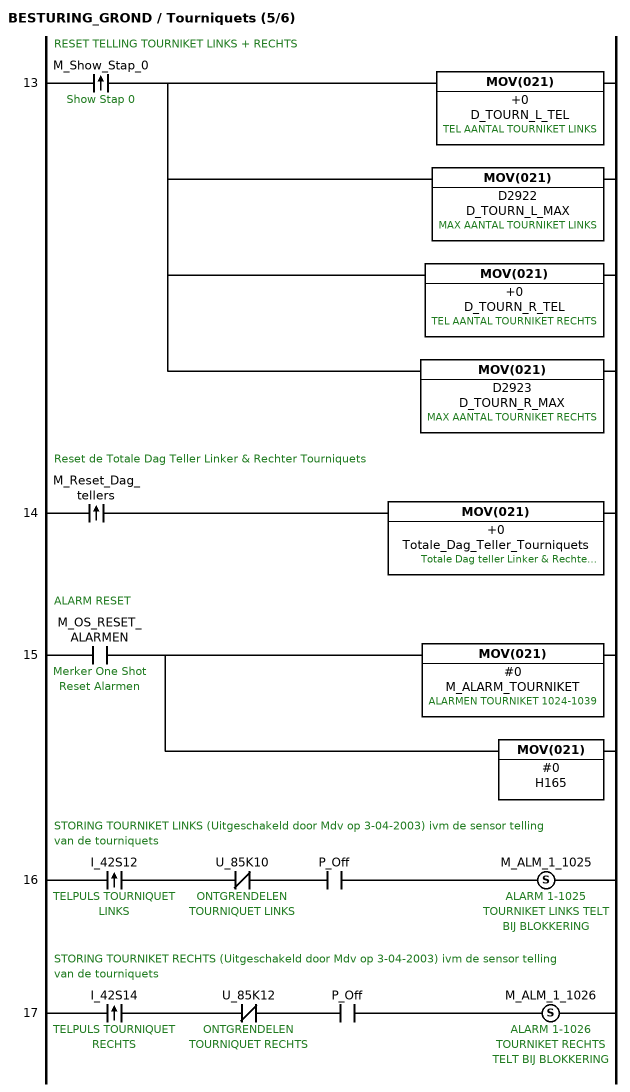
; [picture p144: BESTURING_GROND / Tourniquets, rungs 13-17]
; rung 13: RESET TELLING TOURNIKET LINKS + RECHTS
@LD M_Show_Stap_0  ; Show Stap 0
MOV(021) +0 D_TOURN_L_TEL  ; TEL AANTAL TOURNIKET LINKS
MOV(021) D2922 D_TOURN_L_MAX  ; MAX AANTAL TOURNIKET LINKS
MOV(021) +0 D_TOURN_R_TEL  ; TEL AANTAL TOURNIKET RECHTS
MOV(021) D2923 D_TOURN_R_MAX  ; MAX AANTAL TOURNIKET RECHTS
; rung 14: Reset de Totale Dag Teller Linker & Rechter Tourniquets
@LD M_Reset_Dag_tellers
MOV(021) +0 Totale_Dag_Teller_Tourniquets  ; Totale Dag teller Linker & Rechter Tournoquets
; rung 15: ALARM RESET
LD M_OS_RESET_ALARMEN  ; Merker One Shot Reset Alarmen
MOV(021) #0 M_ALARM_TOURNIKET  ; ALARMEN TOURNIKET 1024-1039
MOV(021) #0 H165
; rung 16: STORING TOURNIKET LINKS (Uitgeschakeld door Mdv op 3-04-2003) ivm de sensor telling van de tourniquets
@LD I_42S12  ; TELPULS TOURNIQUET LINKS
ANDNOT U_85K10  ; ONTGRENDELEN TOURNIQUET LINKS
AND P_Off
SET M_ALM_1_1025  ; ALARM 1-1025 TOURNIKET LINKS TELT BIJ BLOKKERING
; rung 17: STORING TOURNIKET RECHTS (Uitgeschakeld door Mdv op 3-04-2003) ivm de sensor telling van de tourniquets
@LD I_42S14  ; TELPULS TOURNIQUET RECHTS
ANDNOT U_85K12  ; ONTGRENDELEN TOURNIQUET RECHTS
AND P_Off
SET M_ALM_1_1026  ; ALARM 1-1026 TOURNIKET RECHTS TELT BIJ BLOKKERING

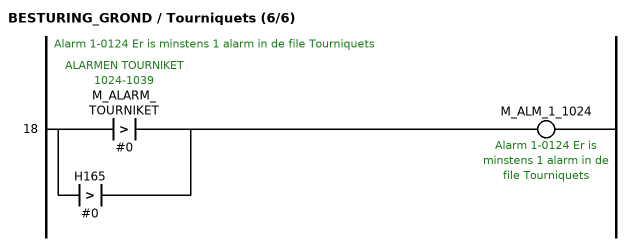
; rung 18: Alarm 1-0124 Er is minstens 1 alarm in de file Tourniquets
LD>(320) M_ALARM_TOURNIKET #0  ; ALARMEN TOURNIKET 1024-1039
OR>(320) H165 #0
OUT M_ALM_1_1024  ; Alarm 1-0124 Er is minstens 1 alarm in de file Tourniquets

### Section Hydaruliek_Arm

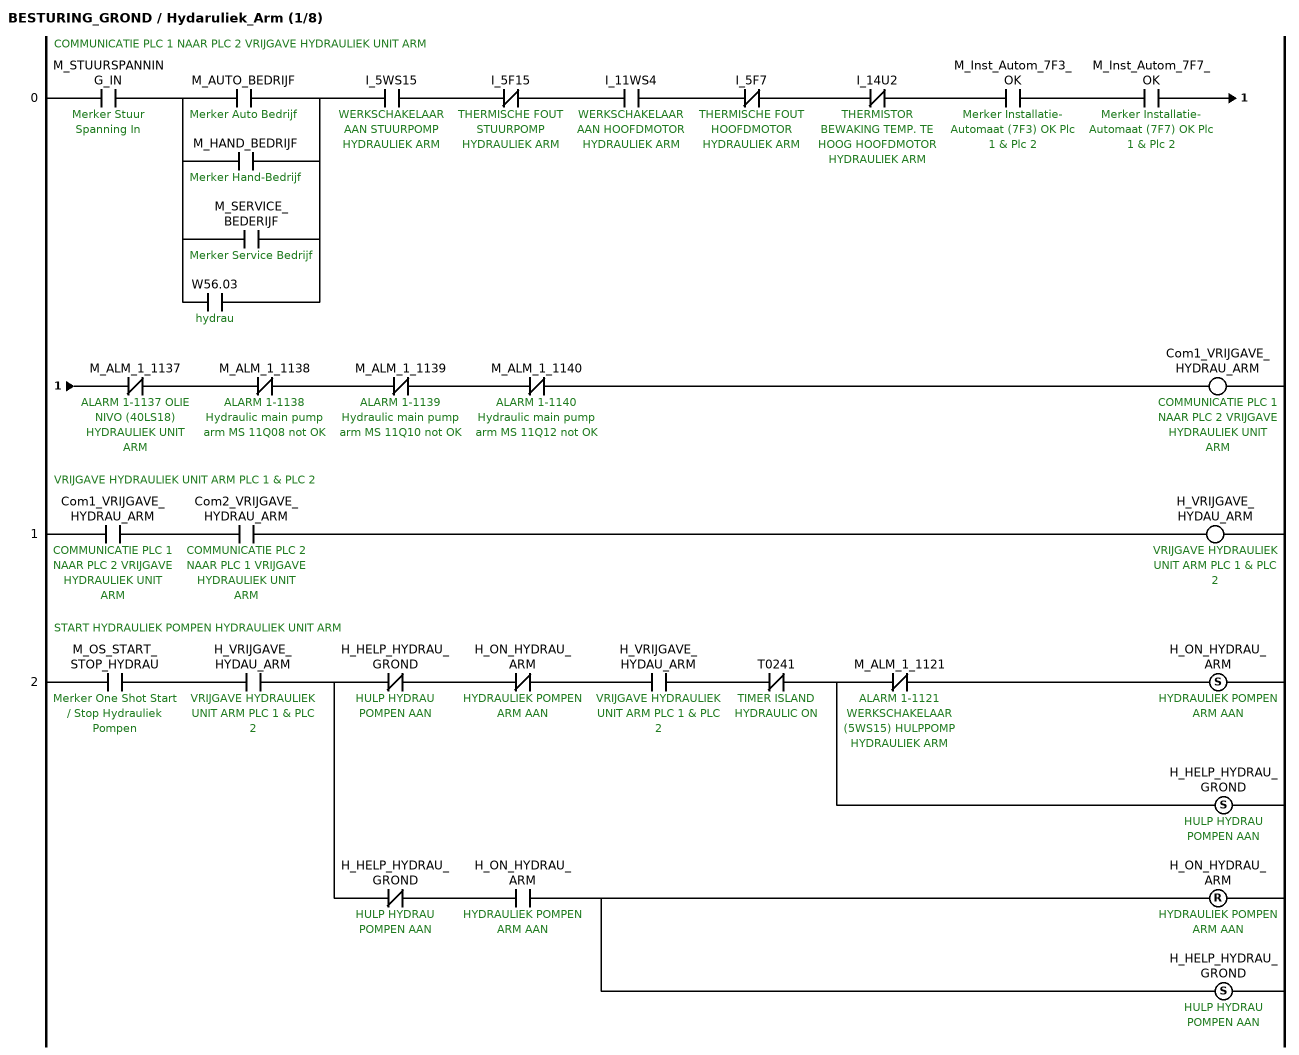
; rung 0: COMMUNICATIE PLC 1 NAAR PLC 2 VRIJGAVE HYDRAULIEK UNIT ARM
LD M_STUURSPANNING_IN  ; Merker Stuur Spanning In
LD M_AUTO_BEDRIJF  ; Merker Auto Bedrijf
OR M_HAND_BEDRIJF  ; Merker Hand-Bedrijf
OR M_SERVICE_BEDERIJF  ; Merker Service Bedrijf
OR W56.03  ; hydrau
ANDLD
AND I_5WS15  ; WERKSCHAKELAAR AAN STUURPOMP HYDRAULIEK ARM
ANDNOT I_5F15  ; THERMISCHE FOUT STUURPOMP HYDRAULIEK ARM
AND I_11WS4  ; WERKSCHAKELAAR AAN HOOFDMOTOR HYDRAULIEK ARM
ANDNOT I_5F7  ; THERMISCHE FOUT HOOFDMOTOR HYDRAULIEK ARM
ANDNOT I_14U2  ; THERMISTOR BEWAKING TEMP. TE HOOG HOOFDMOTOR HYDRAULIEK ARM
AND M_Inst_Autom_7F3_OK  ; Merker Installatie-Automaat (7F3) OK Plc 1 & Plc 2
AND M_Inst_Autom_7F7_OK  ; Merker Installatie-Automaat (7F7) OK Plc 1 & Plc 2
ANDNOT M_ALM_1_1137  ; ALARM 1-1137 OLIE NIVO (40LS18) HYDRAULIEK UNIT ARM
ANDNOT M_ALM_1_1138  ; ALARM 1-1138 Hydraulic main pump arm MS 11Q08 not OK
ANDNOT M_ALM_1_1139  ; ALARM 1-1139 Hydraulic main pump arm MS 11Q10 not OK
ANDNOT M_ALM_1_1140  ; ALARM 1-1140 Hydraulic main pump arm MS 11Q12 not OK
OUT Com1_VRIJGAVE_HYDRAU_ARM  ; COMMUNICATIE PLC 1 NAAR PLC 2 VRIJGAVE HYDRAULIEK UNIT ARM
; rung 1: VRIJGAVE HYDRAULIEK UNIT ARM PLC 1 & PLC 2
LD Com1_VRIJGAVE_HYDRAU_ARM  ; COMMUNICATIE PLC 1 NAAR PLC 2 VRIJGAVE HYDRAULIEK UNIT ARM
AND Com2_VRIJGAVE_HYDRAU_ARM  ; COMMUNICATIE PLC 2 NAAR PLC 1 VRIJGAVE HYDRAULIEK UNIT ARM
OUT H_VRIJGAVE_HYDAU_ARM  ; VRIJGAVE HYDRAULIEK UNIT ARM PLC 1 & PLC 2
; rung 2: START HYDRAULIEK POMPEN HYDRAULIEK UNIT ARM
LD M_OS_START_STOP_HYDRAU  ; Merker One Shot Start / Stop Hydrauliek Pompen
AND H_VRIJGAVE_HYDAU_ARM  ; VRIJGAVE HYDRAULIEK UNIT ARM PLC 1 & PLC 2
OUT TR0
ANDNOT H_HELP_HYDRAU_GROND  ; HULP HYDRAU POMPEN AAN
ANDNOT H_ON_HYDRAU_ARM  ; HYDRAULIEK POMPEN ARM AAN
AND H_VRIJGAVE_HYDAU_ARM  ; VRIJGAVE HYDRAULIEK UNIT ARM PLC 1 & PLC 2
ANDNOT T0241  ; TIMER ISLAND HYDRAULIC ON
OUT TR1
ANDNOT M_ALM_1_1121  ; ALARM 1-1121 WERKSCHAKELAAR (5WS15) HULPPOMP HYDRAULIEK ARM
SET H_ON_HYDRAU_ARM  ; HYDRAULIEK POMPEN ARM AAN
LD TR1
SET H_HELP_HYDRAU_GROND  ; HULP HYDRAU POMPEN AAN
LD TR0
ANDNOT H_HELP_HYDRAU_GROND  ; HULP HYDRAU POMPEN AAN
AND H_ON_HYDRAU_ARM  ; HYDRAULIEK POMPEN ARM AAN
RSET H_ON_HYDRAU_ARM  ; HYDRAULIEK POMPEN ARM AAN
SET H_HELP_HYDRAU_GROND  ; HULP HYDRAU POMPEN AAN

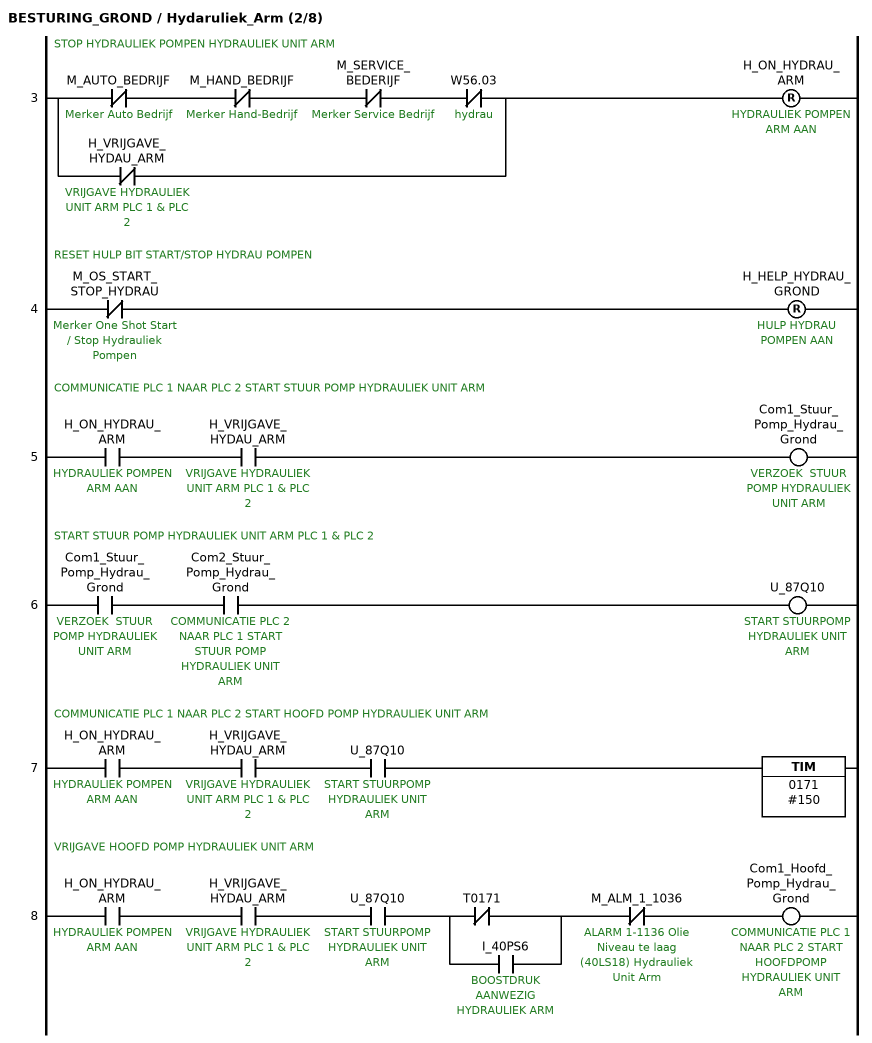
; rung 3: STOP HYDRAULIEK POMPEN HYDRAULIEK UNIT ARM
LDNOT M_AUTO_BEDRIJF  ; Merker Auto Bedrijf
ANDNOT M_HAND_BEDRIJF  ; Merker Hand-Bedrijf
ANDNOT M_SERVICE_BEDERIJF  ; Merker Service Bedrijf
ANDNOT W56.03  ; hydrau
ORNOT H_VRIJGAVE_HYDAU_ARM  ; VRIJGAVE HYDRAULIEK UNIT ARM PLC 1 & PLC 2
RSET H_ON_HYDRAU_ARM  ; HYDRAULIEK POMPEN ARM AAN
; rung 4: RESET HULP BIT START/STOP HYDRAU POMPEN
LDNOT M_OS_START_STOP_HYDRAU  ; Merker One Shot Start / Stop Hydrauliek Pompen
RSET H_HELP_HYDRAU_GROND  ; HULP HYDRAU POMPEN AAN
; rung 5: COMMUNICATIE PLC 1 NAAR PLC 2 START STUUR POMP HYDRAULIEK UNIT ARM
LD H_ON_HYDRAU_ARM  ; HYDRAULIEK POMPEN ARM AAN
AND H_VRIJGAVE_HYDAU_ARM  ; VRIJGAVE HYDRAULIEK UNIT ARM PLC 1 & PLC 2
OUT Com1_Stuur_Pomp_Hydrau_Grond  ; VERZOEK  STUUR POMP HYDRAULIEK UNIT ARM
; rung 6: START STUUR POMP HYDRAULIEK UNIT ARM PLC 1 & PLC 2
LD Com1_Stuur_Pomp_Hydrau_Grond  ; VERZOEK  STUUR POMP HYDRAULIEK UNIT ARM
AND Com2_Stuur_Pomp_Hydrau_Grond  ; COMMUNICATIE PLC 2 NAAR PLC 1 START STUUR POMP HYDRAULIEK UNIT ARM
OUT U_87Q10  ; START STUURPOMP HYDRAULIEK UNIT ARM
; rung 7: COMMUNICATIE PLC 1 NAAR PLC 2 START HOOFD POMP HYDRAULIEK UNIT ARM
LD H_ON_HYDRAU_ARM  ; HYDRAULIEK POMPEN ARM AAN
AND H_VRIJGAVE_HYDAU_ARM  ; VRIJGAVE HYDRAULIEK UNIT ARM PLC 1 & PLC 2
AND U_87Q10  ; START STUURPOMP HYDRAULIEK UNIT ARM
TIM 0171 #150
; rung 8: VRIJGAVE HOOFD POMP HYDRAULIEK UNIT ARM
LD H_ON_HYDRAU_ARM  ; HYDRAULIEK POMPEN ARM AAN
AND H_VRIJGAVE_HYDAU_ARM  ; VRIJGAVE HYDRAULIEK UNIT ARM PLC 1 & PLC 2
AND U_87Q10  ; START STUURPOMP HYDRAULIEK UNIT ARM
LDNOT T0171
OR I_40PS6  ; BOOSTDRUK AANWEZIG HYDRAULIEK ARM
ANDLD
ANDNOT M_ALM_1_1036  ; ALARM 1-1136 Olie Niveau te laag (40LS18) Hydrauliek Unit Arm
OUT Com1_Hoofd_Pomp_Hydrau_Grond  ; COMMUNICATIE PLC 1 NAAR PLC 2 START HOOFDPOMP HYDRAULIEK UNIT ARM

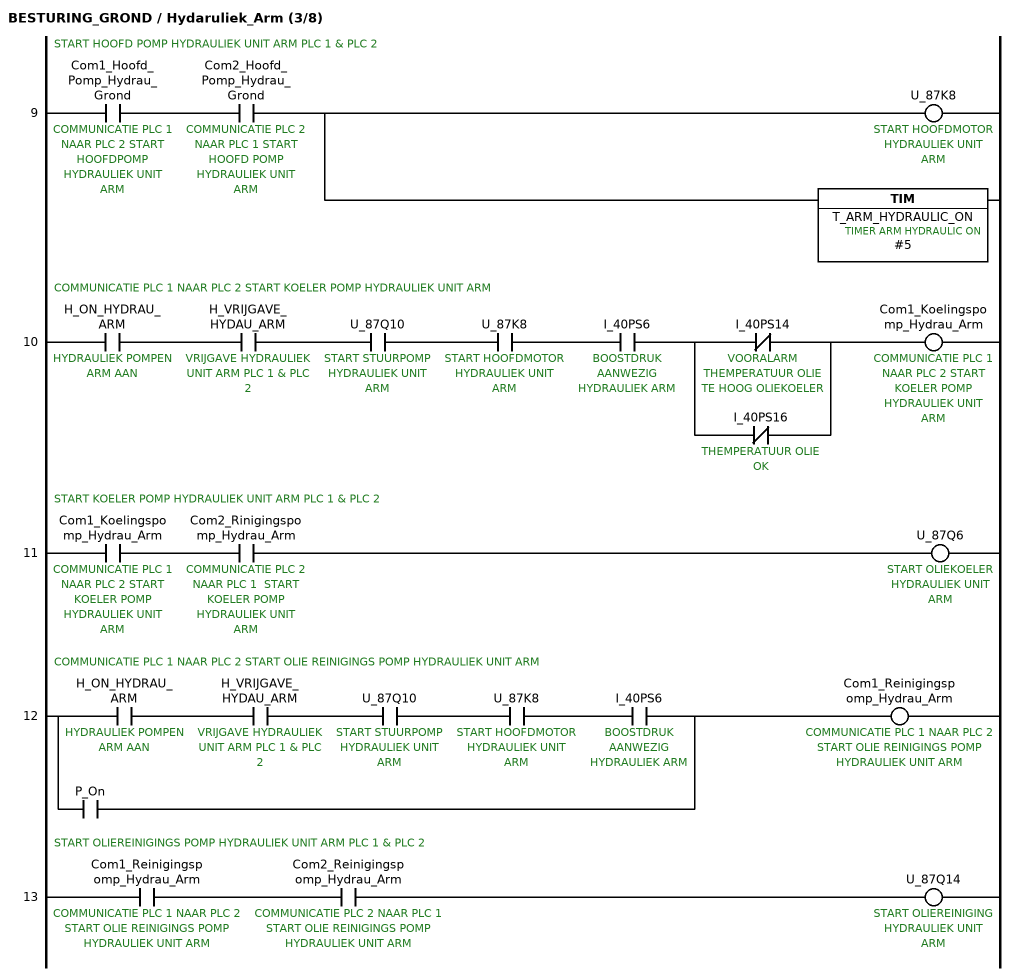
; rung 9: START HOOFD POMP HYDRAULIEK UNIT ARM PLC 1 & PLC 2
LD Com1_Hoofd_Pomp_Hydrau_Grond  ; COMMUNICATIE PLC 1 NAAR PLC 2 START HOOFDPOMP HYDRAULIEK UNIT ARM
AND Com2_Hoofd_Pomp_Hydrau_Grond  ; COMMUNICATIE PLC 2 NAAR PLC 1 START HOOFD POMP HYDRAULIEK UNIT ARM
OUT U_87K8  ; START HOOFDMOTOR HYDRAULIEK UNIT ARM
TIM T_ARM_HYDRAULIC_ON #5  ; TIMER ARM HYDRAULIC ON
; rung 10: COMMUNICATIE PLC 1 NAAR PLC 2 START KOELER POMP HYDRAULIEK UNIT ARM
LD H_ON_HYDRAU_ARM  ; HYDRAULIEK POMPEN ARM AAN
AND H_VRIJGAVE_HYDAU_ARM  ; VRIJGAVE HYDRAULIEK UNIT ARM PLC 1 & PLC 2
AND U_87Q10  ; START STUURPOMP HYDRAULIEK UNIT ARM
AND U_87K8  ; START HOOFDMOTOR HYDRAULIEK UNIT ARM
AND I_40PS6  ; BOOSTDRUK AANWEZIG HYDRAULIEK ARM
LDNOT I_40PS14  ; VOORALARM THEMPERATUUR OLIE TE HOOG OLIEKOELER
ORNOT I_40PS16  ; THEMPERATUUR OLIE OK
ANDLD
OUT Com1_Koelingspomp_Hydrau_Arm  ; COMMUNICATIE PLC 1 NAAR PLC 2 START KOELER POMP HYDRAULIEK UNIT ARM
; rung 11: START KOELER POMP HYDRAULIEK UNIT ARM PLC 1 & PLC 2
LD Com1_Koelingspomp_Hydrau_Arm  ; COMMUNICATIE PLC 1 NAAR PLC 2 START KOELER POMP HYDRAULIEK UNIT ARM
AND Com2_Rinigingspomp_Hydrau_Arm  ; COMMUNICATIE PLC 2 NAAR PLC 1  START KOELER POMP HYDRAULIEK UNIT ARM
OUT U_87Q6  ; START OLIEKOELER HYDRAULIEK UNIT ARM
; rung 12: COMMUNICATIE PLC 1 NAAR PLC 2 START OLIE REINIGINGS POMP HYDRAULIEK UNIT ARM
LD H_ON_HYDRAU_ARM  ; HYDRAULIEK POMPEN ARM AAN
AND H_VRIJGAVE_HYDAU_ARM  ; VRIJGAVE HYDRAULIEK UNIT ARM PLC 1 & PLC 2
AND U_87Q10  ; START STUURPOMP HYDRAULIEK UNIT ARM
AND U_87K8  ; START HOOFDMOTOR HYDRAULIEK UNIT ARM
AND I_40PS6  ; BOOSTDRUK AANWEZIG HYDRAULIEK ARM
OR P_On
OUT Com1_Reinigingspomp_Hydrau_Arm  ; COMMUNICATIE PLC 1 NAAR PLC 2 START OLIE REINIGINGS POMP HYDRAULIEK UNIT ARM
; rung 13: START OLIEREINIGINGS POMP HYDRAULIEK UNIT ARM PLC 1 & PLC 2
LD Com1_Reinigingspomp_Hydrau_Arm  ; COMMUNICATIE PLC 1 NAAR PLC 2 START OLIE REINIGINGS POMP HYDRAULIEK UNIT ARM
AND Com2_Reinigingspomp_Hydrau_Arm  ; COMMUNICATIE PLC 2 NAAR PLC 1 START OLIE REINIGINGS POMP HYDRAULIEK UNIT ARM
OUT U_87Q14  ; START OLIEREINIGING HYDRAULIEK UNIT ARM

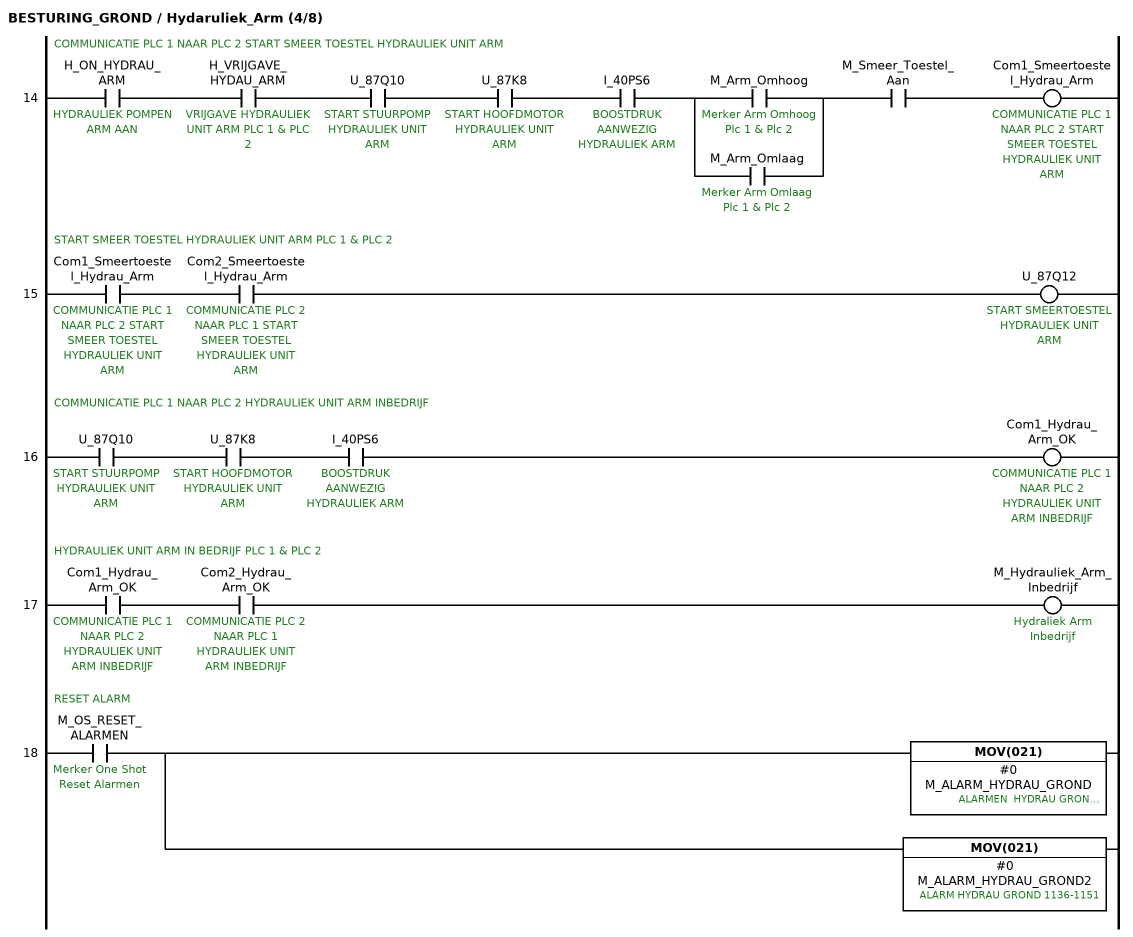
; rung 14: COMMUNICATIE PLC 1 NAAR PLC 2 START SMEER TOESTEL HYDRAULIEK UNIT ARM
LD H_ON_HYDRAU_ARM  ; HYDRAULIEK POMPEN ARM AAN
AND H_VRIJGAVE_HYDAU_ARM  ; VRIJGAVE HYDRAULIEK UNIT ARM PLC 1 & PLC 2
AND U_87Q10  ; START STUURPOMP HYDRAULIEK UNIT ARM
AND U_87K8  ; START HOOFDMOTOR HYDRAULIEK UNIT ARM
AND I_40PS6  ; BOOSTDRUK AANWEZIG HYDRAULIEK ARM
LD M_Arm_Omhoog  ; Merker Arm Omhoog Plc 1 & Plc 2
OR M_Arm_Omlaag  ; Merker Arm Omlaag Plc 1 & Plc 2
ANDLD
AND M_Smeer_Toestel_Aan
OUT Com1_Smeertoestel_Hydrau_Arm  ; COMMUNICATIE PLC 1 NAAR PLC 2 START SMEER TOESTEL HYDRAULIEK UNIT ARM
; rung 15: START SMEER TOESTEL HYDRAULIEK UNIT ARM PLC 1 & PLC 2
LD Com1_Smeertoestel_Hydrau_Arm  ; COMMUNICATIE PLC 1 NAAR PLC 2 START SMEER TOESTEL HYDRAULIEK UNIT ARM
AND Com2_Smeertoestel_Hydrau_Arm  ; COMMUNICATIE PLC 2 NAAR PLC 1 START SMEER TOESTEL HYDRAULIEK UNIT ARM
OUT U_87Q12  ; START SMEERTOESTEL HYDRAULIEK UNIT ARM
; rung 16: COMMUNICATIE PLC 1 NAAR PLC 2 HYDRAULIEK UNIT ARM INBEDRIJF
LD U_87Q10  ; START STUURPOMP HYDRAULIEK UNIT ARM
AND U_87K8  ; START HOOFDMOTOR HYDRAULIEK UNIT ARM
AND I_40PS6  ; BOOSTDRUK AANWEZIG HYDRAULIEK ARM
OUT Com1_Hydrau_Arm_OK  ; COMMUNICATIE PLC 1 NAAR PLC 2 HYDRAULIEK UNIT ARM INBEDRIJF
; rung 17: HYDRAULIEK UNIT ARM IN BEDRIJF PLC 1 & PLC 2
LD Com1_Hydrau_Arm_OK  ; COMMUNICATIE PLC 1 NAAR PLC 2 HYDRAULIEK UNIT ARM INBEDRIJF
AND Com2_Hydrau_Arm_OK  ; COMMUNICATIE PLC 2 NAAR PLC 1 HYDRAULIEK UNIT ARM INBEDRIJF
OUT M_Hydrauliek_Arm_Inbedrijf  ; Hydraliek Arm Inbedrijf
; rung 18: RESET ALARM
LD M_OS_RESET_ALARMEN  ; Merker One Shot Reset Alarmen
MOV(021) #0 M_ALARM_HYDRAU_GROND  ; ALARMEN  HYDRAU GROND 1120-1135
MOV(021) #0 M_ALARM_HYDRAU_GROND2  ; ALARM HYDRAU GROND 1136-1151

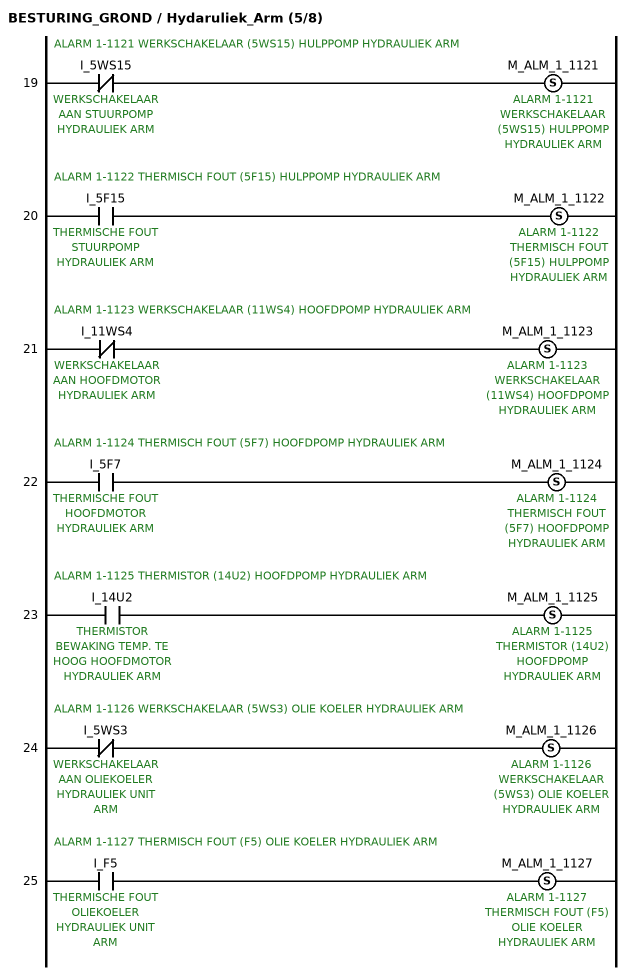
; rung 19: ALARM 1-1121 WERKSCHAKELAAR (5WS15) HULPPOMP HYDRAULIEK ARM
LDNOT I_5WS15  ; WERKSCHAKELAAR AAN STUURPOMP HYDRAULIEK ARM
SET M_ALM_1_1121  ; ALARM 1-1121 WERKSCHAKELAAR (5WS15) HULPPOMP HYDRAULIEK ARM
; rung 20: ALARM 1-1122 THERMISCH FOUT (5F15) HULPPOMP HYDRAULIEK ARM
LD I_5F15  ; THERMISCHE FOUT STUURPOMP HYDRAULIEK ARM
SET M_ALM_1_1122  ; ALARM 1-1122 THERMISCH FOUT (5F15) HULPPOMP HYDRAULIEK ARM
; rung 21: ALARM 1-1123 WERKSCHAKELAAR (11WS4) HOOFDPOMP HYDRAULIEK ARM
LDNOT I_11WS4  ; WERKSCHAKELAAR AAN HOOFDMOTOR HYDRAULIEK ARM
SET M_ALM_1_1123  ; ALARM 1-1123 WERKSCHAKELAAR (11WS4) HOOFDPOMP HYDRAULIEK ARM
; rung 22: ALARM 1-1124 THERMISCH FOUT (5F7) HOOFDPOMP HYDRAULIEK ARM
LD I_5F7  ; THERMISCHE FOUT HOOFDMOTOR HYDRAULIEK ARM
SET M_ALM_1_1124  ; ALARM 1-1124 THERMISCH FOUT (5F7) HOOFDPOMP HYDRAULIEK ARM
; rung 23: ALARM 1-1125 THERMISTOR (14U2) HOOFDPOMP HYDRAULIEK ARM
LD I_14U2  ; THERMISTOR BEWAKING TEMP. TE HOOG HOOFDMOTOR HYDRAULIEK ARM
SET M_ALM_1_1125  ; ALARM 1-1125 THERMISTOR (14U2) HOOFDPOMP HYDRAULIEK ARM
; rung 24: ALARM 1-1126 WERKSCHAKELAAR (5WS3) OLIE KOELER HYDRAULIEK ARM
LDNOT I_5WS3  ; WERKSCHAKELAAR AAN OLIEKOELER HYDRAULIEK UNIT ARM
SET M_ALM_1_1126  ; ALARM 1-1126 WERKSCHAKELAAR (5WS3) OLIE KOELER HYDRAULIEK ARM
; rung 25: ALARM 1-1127 THERMISCH FOUT (F5) OLIE KOELER HYDRAULIEK ARM
LD I_F5  ; THERMISCHE FOUT OLIEKOELER HYDRAULIEK UNIT ARM
SET M_ALM_1_1127  ; ALARM 1-1127 THERMISCH FOUT (F5) OLIE KOELER HYDRAULIEK ARM

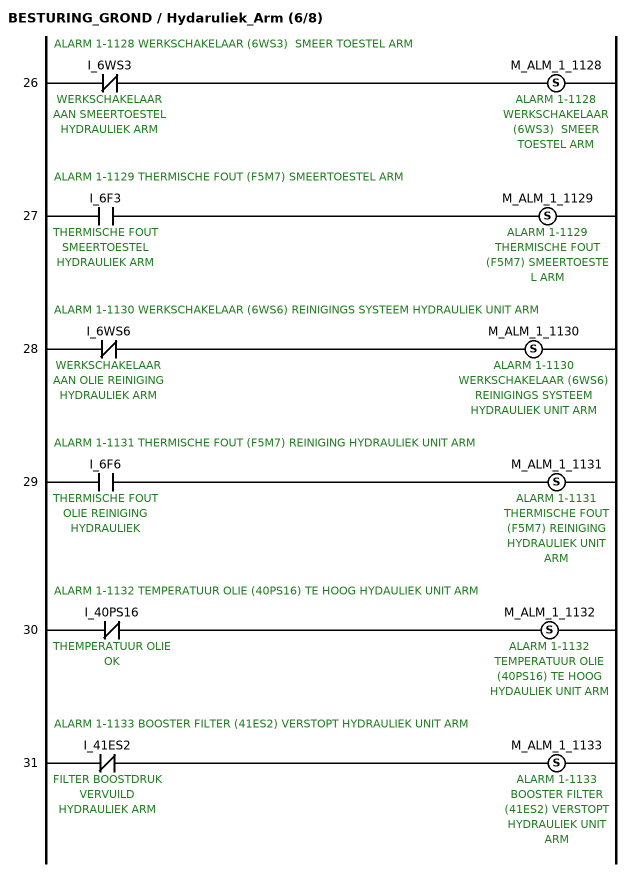
; rung 26: ALARM 1-1128 WERKSCHAKELAAR (6WS3)  SMEER TOESTEL ARM
LDNOT I_6WS3  ; WERKSCHAKELAAR AAN SMEERTOESTEL HYDRAULIEK ARM
SET M_ALM_1_1128  ; ALARM 1-1128 WERKSCHAKELAAR (6WS3)  SMEER TOESTEL ARM
; rung 27: ALARM 1-1129 THERMISCHE FOUT (F5M7) SMEERTOESTEL ARM
LD I_6F3  ; THERMISCHE FOUT SMEERTOESTEL HYDRAULIEK ARM
SET M_ALM_1_1129  ; ALARM 1-1129 THERMISCHE FOUT (F5M7) SMEERTOESTEL ARM
; rung 28: ALARM 1-1130 WERKSCHAKELAAR (6WS6) REINIGINGS SYSTEEM HYDRAULIEK UNIT ARM
LDNOT I_6WS6  ; WERKSCHAKELAAR AAN OLIE REINIGING HYDRAULIEK ARM
SET M_ALM_1_1130  ; ALARM 1-1130 WERKSCHAKELAAR (6WS6) REINIGINGS SYSTEEM HYDRAULIEK UNIT ARM
; rung 29: ALARM 1-1131 THERMISCHE FOUT (F5M7) REINIGING HYDRAULIEK UNIT ARM
LD I_6F6  ; THERMISCHE FOUT OLIE REINIGING HYDRAULIEK
SET M_ALM_1_1131  ; ALARM 1-1131 THERMISCHE FOUT (F5M7) REINIGING HYDRAULIEK UNIT ARM
; rung 30: ALARM 1-1132 TEMPERATUUR OLIE (40PS16) TE HOOG HYDAULIEK UNIT ARM
LDNOT I_40PS16  ; THEMPERATUUR OLIE OK
SET M_ALM_1_1132  ; ALARM 1-1132 TEMPERATUUR OLIE (40PS16) TE HOOG HYDAULIEK UNIT ARM
; rung 31: ALARM 1-1133 BOOSTER FILTER (41ES2) VERSTOPT HYDRAULIEK UNIT ARM
LDNOT I_41ES2  ; FILTER BOOSTDRUK VERVUILD HYDRAULIEK ARM
SET M_ALM_1_1133  ; ALARM 1-1133 BOOSTER FILTER (41ES2) VERSTOPT HYDRAULIEK UNIT ARM

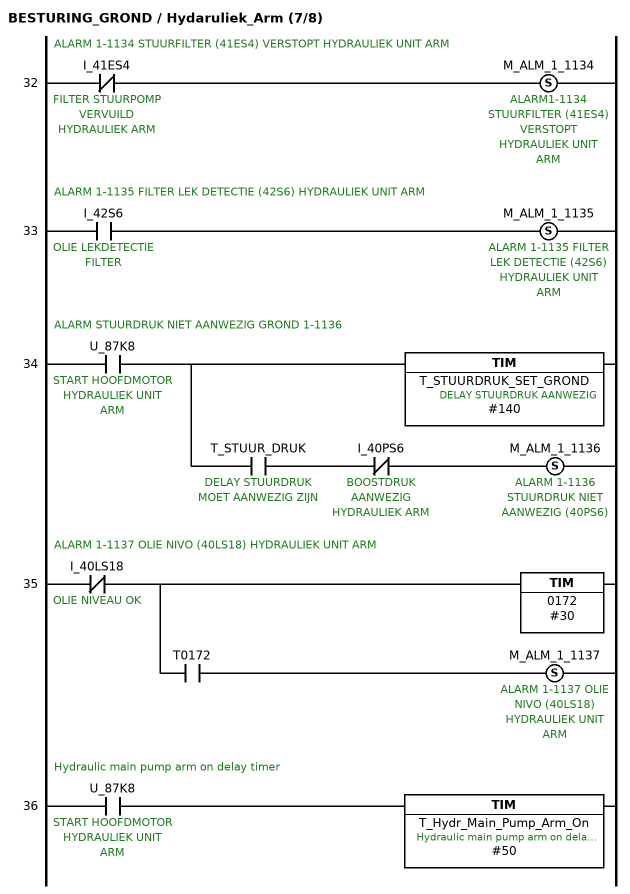
; rung 32: ALARM 1-1134 STUURFILTER (41ES4) VERSTOPT HYDRAULIEK UNIT ARM
LDNOT I_41ES4  ; FILTER STUURPOMP VERVUILD HYDRAULIEK ARM
SET M_ALM_1_1134  ; ALARM1-1134 STUURFILTER (41ES4) VERSTOPT HYDRAULIEK UNIT ARM
; rung 33: ALARM 1-1135 FILTER LEK DETECTIE (42S6) HYDRAULIEK UNIT ARM
LD I_42S6  ; OLIE LEKDETECTIE FILTER
SET M_ALM_1_1135  ; ALARM 1-1135 FILTER LEK DETECTIE (42S6) HYDRAULIEK UNIT ARM
; rung 34: ALARM STUURDRUK NIET AANWEZIG GROND 1-1136
LD U_87K8  ; START HOOFDMOTOR HYDRAULIEK UNIT ARM
TIM T_STUURDRUK_SET_GROND #140  ; DELAY STUURDRUK AANWEZIG
AND T_STUUR_DRUK  ; DELAY STUURDRUK MOET AANWEZIG ZIJN
ANDNOT I_40PS6  ; BOOSTDRUK AANWEZIG HYDRAULIEK ARM
SET M_ALM_1_1136  ; ALARM 1-1136 STUURDRUK NIET AANWEZIG (40PS6)
; rung 35: ALARM 1-1137 OLIE NIVO (40LS18) HYDRAULIEK UNIT ARM
LDNOT I_40LS18  ; OLIE NIVEAU OK
TIM 0172 #30
AND T0172
SET M_ALM_1_1137  ; ALARM 1-1137 OLIE NIVO (40LS18) HYDRAULIEK UNIT ARM
; rung 36: Hydraulic main pump arm on delay timer
LD U_87K8  ; START HOOFDMOTOR HYDRAULIEK UNIT ARM
TIM T_Hydr_Main_Pump_Arm_On #50  ; Hydraulic main pump arm on delay timer

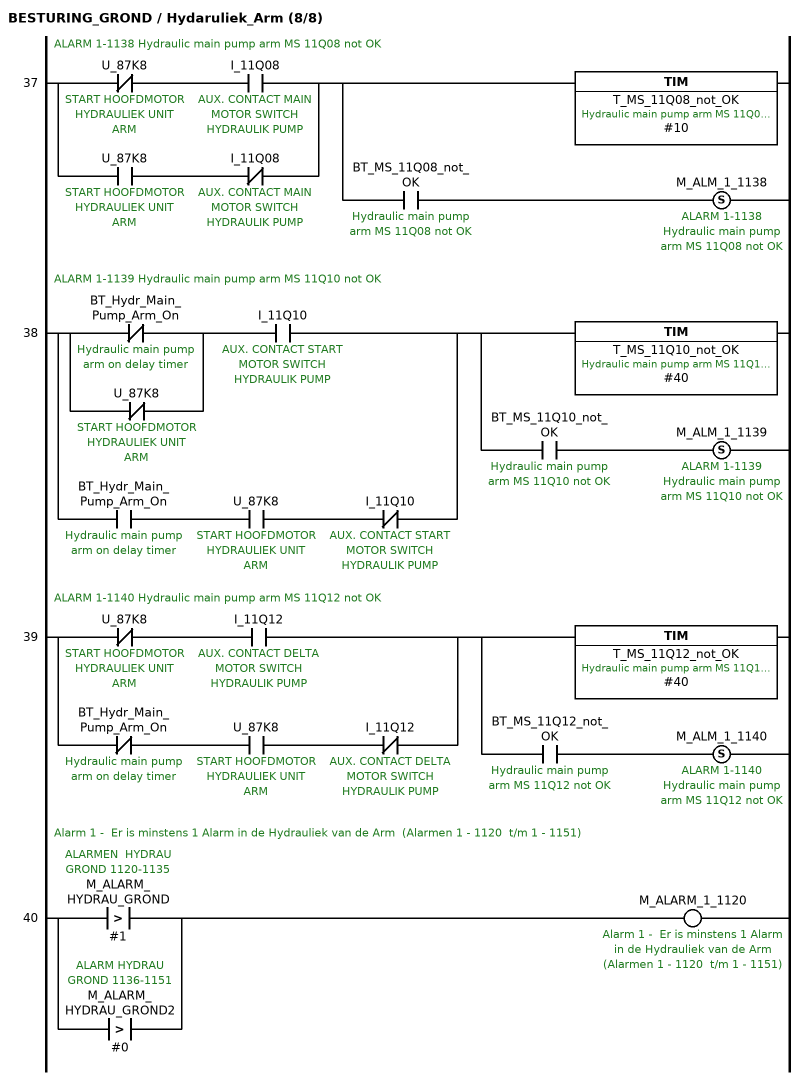
; rung 37: ALARM 1-1138 Hydraulic main pump arm MS 11Q08 not OK
LDNOT U_87K8  ; START HOOFDMOTOR HYDRAULIEK UNIT ARM
AND I_11Q08  ; AUX. CONTACT MAIN MOTOR SWITCH HYDRAULIK PUMP
LD U_87K8  ; START HOOFDMOTOR HYDRAULIEK UNIT ARM
ANDNOT I_11Q08  ; AUX. CONTACT MAIN MOTOR SWITCH HYDRAULIK PUMP
ORLD
TIM T_MS_11Q08_not_OK #10  ; Hydraulic main pump arm MS 11Q08 not OK
AND BT_MS_11Q08_not_OK  ; Hydraulic main pump arm MS 11Q08 not OK
SET M_ALM_1_1138  ; ALARM 1-1138 Hydraulic main pump arm MS 11Q08 not OK
; rung 38: ALARM 1-1139 Hydraulic main pump arm MS 11Q10 not OK
LDNOT BT_Hydr_Main_Pump_Arm_On  ; Hydraulic main pump arm on delay timer
ORNOT U_87K8  ; START HOOFDMOTOR HYDRAULIEK UNIT ARM
AND I_11Q10  ; AUX. CONTACT START MOTOR SWITCH HYDRAULIK PUMP
LD BT_Hydr_Main_Pump_Arm_On  ; Hydraulic main pump arm on delay timer
AND U_87K8  ; START HOOFDMOTOR HYDRAULIEK UNIT ARM
ANDNOT I_11Q10  ; AUX. CONTACT START MOTOR SWITCH HYDRAULIK PUMP
ORLD
TIM T_MS_11Q10_not_OK #40  ; Hydraulic main pump arm MS 11Q10 not OK
AND BT_MS_11Q10_not_OK  ; Hydraulic main pump arm MS 11Q10 not OK
SET M_ALM_1_1139  ; ALARM 1-1139 Hydraulic main pump arm MS 11Q10 not OK
; rung 39: ALARM 1-1140 Hydraulic main pump arm MS 11Q12 not OK
LDNOT U_87K8  ; START HOOFDMOTOR HYDRAULIEK UNIT ARM
AND I_11Q12  ; AUX. CONTACT DELTA MOTOR SWITCH HYDRAULIK PUMP
LDNOT BT_Hydr_Main_Pump_Arm_On  ; Hydraulic main pump arm on delay timer
AND U_87K8  ; START HOOFDMOTOR HYDRAULIEK UNIT ARM
ANDNOT I_11Q12  ; AUX. CONTACT DELTA MOTOR SWITCH HYDRAULIK PUMP
ORLD
TIM T_MS_11Q12_not_OK #40  ; Hydraulic main pump arm MS 11Q12 not OK
AND BT_MS_11Q12_not_OK  ; Hydraulic main pump arm MS 11Q12 not OK
SET M_ALM_1_1140  ; ALARM 1-1140 Hydraulic main pump arm MS 11Q12 not OK
; rung 40: Alarm 1 -  Er is minstens 1 Alarm in de Hydrauliek van de Arm  (Alarmen 1 - 1120  t/m 1 - 1151)
LD>(320) M_ALARM_HYDRAU_GROND #1  ; ALARMEN  HYDRAU GROND 1120-1135
OR>(320) M_ALARM_HYDRAU_GROND2 #0  ; ALARM HYDRAU GROND 1136-1151
OUT M_ALARM_1_1120  ; Alarm 1 -  Er is minstens 1 Alarm in de Hydrauliek van de Arm  (Alarmen 1 - 1120  t/m 1 - 1151)

### Section Data_Arm

### Section Besturing_Arm

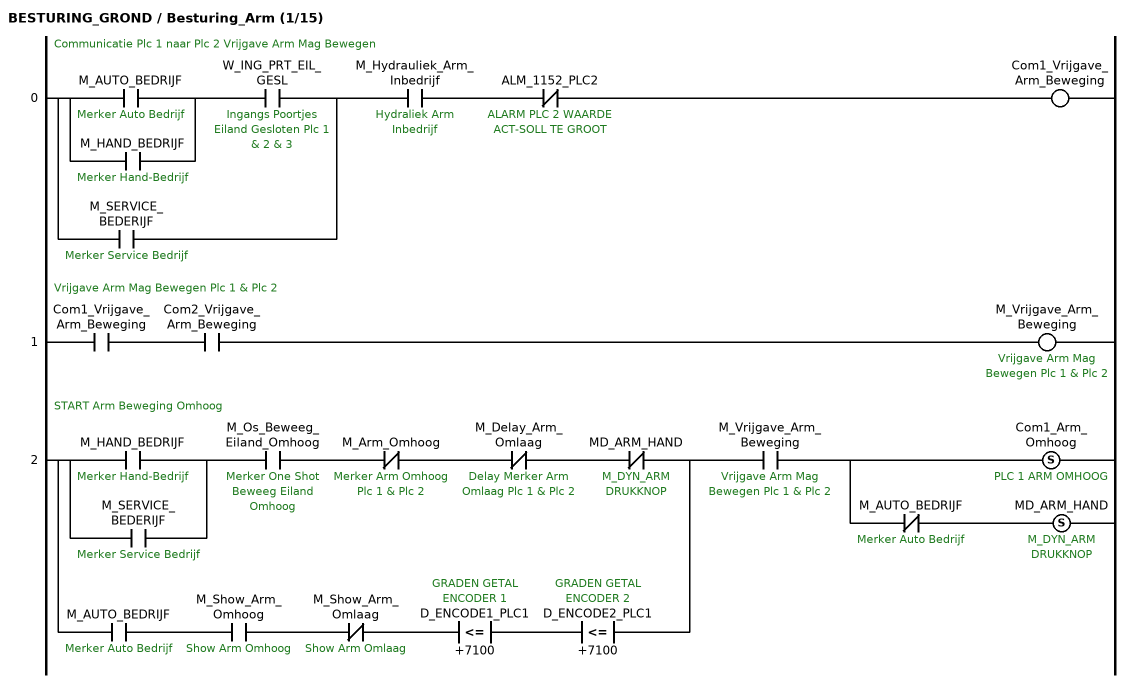
; rung 0: Communicatie Plc 1 naar Plc 2 Vrijgave Arm Mag Bewegen
LD M_AUTO_BEDRIJF  ; Merker Auto Bedrijf
OR M_HAND_BEDRIJF  ; Merker Hand-Bedrijf
AND W_ING_PRT_EIL_GESL  ; Ingangs Poortjes Eiland Gesloten Plc 1 & 2 & 3
OR M_SERVICE_BEDERIJF  ; Merker Service Bedrijf
AND M_Hydrauliek_Arm_Inbedrijf  ; Hydraliek Arm Inbedrijf
ANDNOT ALM_1152_PLC2  ; ALARM PLC 2 WAARDE ACT-SOLL TE GROOT
OUT Com1_Vrijgave_Arm_Beweging
; rung 1: Vrijgave Arm Mag Bewegen Plc 1 & Plc 2
LD Com1_Vrijgave_Arm_Beweging
AND Com2_Vrijgave_Arm_Beweging
OUT M_Vrijgave_Arm_Beweging  ; Vrijgave Arm Mag Bewegen Plc 1 & Plc 2
; rung 2: START Arm Beweging Omhoog
LD M_HAND_BEDRIJF  ; Merker Hand-Bedrijf
OR M_SERVICE_BEDERIJF  ; Merker Service Bedrijf
AND M_Os_Beweeg_Eiland_Omhoog  ; Merker One Shot Beweeg Eiland Omhoog
ANDNOT M_Arm_Omhoog  ; Merker Arm Omhoog Plc 1 & Plc 2
ANDNOT M_Delay_Arm_Omlaag  ; Delay Merker Arm Omlaag Plc 1 & Plc 2
ANDNOT MD_ARM_HAND  ; M_DYN_ARM DRUKKNOP
LD M_AUTO_BEDRIJF  ; Merker Auto Bedrijf
AND M_Show_Arm_Omhoog  ; Show Arm Omhoog
ANDNOT M_Show_Arm_Omlaag  ; Show Arm Omlaag
AND<=S(317) D_ENCODE1_PLC1 +7100  ; GRADEN GETAL ENCODER 1
AND<=S(317) D_ENCODE2_PLC1 +7100  ; GRADEN GETAL ENCODER 2
ORLD
AND M_Vrijgave_Arm_Beweging  ; Vrijgave Arm Mag Bewegen Plc 1 & Plc 2
SET Com1_Arm_Omhoog  ; PLC 1 ARM OMHOOG
ANDNOT M_AUTO_BEDRIJF  ; Merker Auto Bedrijf
SET MD_ARM_HAND  ; M_DYN_ARM DRUKKNOP

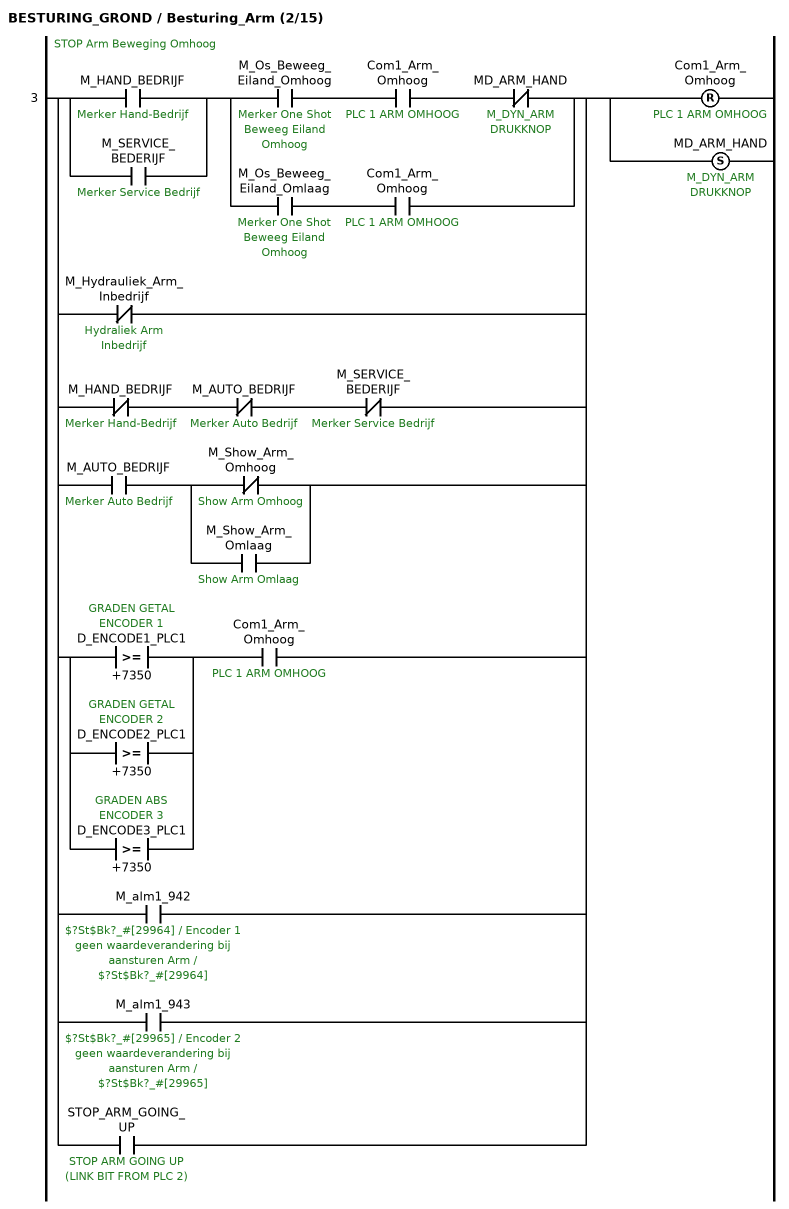
; rung 3: STOP Arm Beweging Omhoog
LD M_HAND_BEDRIJF  ; Merker Hand-Bedrijf
OR M_SERVICE_BEDERIJF  ; Merker Service Bedrijf
LD M_Os_Beweeg_Eiland_Omhoog  ; Merker One Shot Beweeg Eiland Omhoog
AND Com1_Arm_Omhoog  ; PLC 1 ARM OMHOOG
ANDNOT MD_ARM_HAND  ; M_DYN_ARM DRUKKNOP
LD M_Os_Beweeg_Eiland_Omlaag  ; Merker One Shot Beweeg Eiland Omhoog
AND Com1_Arm_Omhoog  ; PLC 1 ARM OMHOOG
ORLD
ANDLD
ORNOT M_Hydrauliek_Arm_Inbedrijf  ; Hydraliek Arm Inbedrijf
LDNOT M_HAND_BEDRIJF  ; Merker Hand-Bedrijf
ANDNOT M_AUTO_BEDRIJF  ; Merker Auto Bedrijf
ANDNOT M_SERVICE_BEDERIJF  ; Merker Service Bedrijf
ORLD
LD M_AUTO_BEDRIJF  ; Merker Auto Bedrijf
LDNOT M_Show_Arm_Omhoog  ; Show Arm Omhoog
OR M_Show_Arm_Omlaag  ; Show Arm Omlaag
ANDLD
ORLD
LD>=S(327) D_ENCODE1_PLC1 +7350  ; GRADEN GETAL ENCODER 1
OR>=S(327) D_ENCODE2_PLC1 +7350  ; GRADEN GETAL ENCODER 2
OR>=S(327) D_ENCODE3_PLC1 +7350  ; GRADEN ABS ENCODER 3
AND Com1_Arm_Omhoog  ; PLC 1 ARM OMHOOG
ORLD
OR M_alm1_942  ; $?St$Bk?_#[29964] / Encoder 1 geen waardeverandering bij aansturen Arm / $?St$Bk?_#[29964]
OR M_alm1_943  ; $?St$Bk?_#[29965] / Encoder 2 geen waardeverandering bij aansturen Arm / $?St$Bk?_#[29965]
OR STOP_ARM_GOING_UP  ; STOP ARM GOING UP (LINK BIT FROM PLC 2)
RSET Com1_Arm_Omhoog  ; PLC 1 ARM OMHOOG
SET MD_ARM_HAND  ; M_DYN_ARM DRUKKNOP

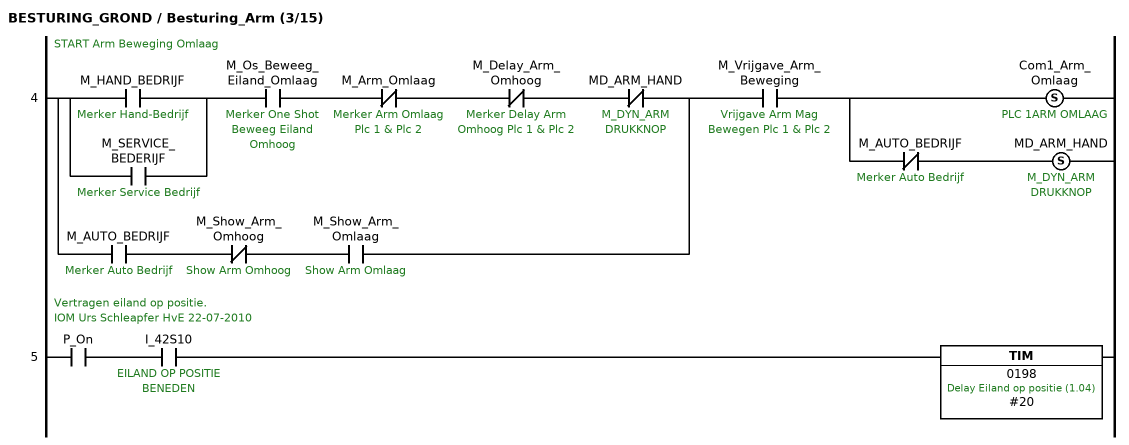
; rung 4: START Arm Beweging Omlaag
LD M_HAND_BEDRIJF  ; Merker Hand-Bedrijf
OR M_SERVICE_BEDERIJF  ; Merker Service Bedrijf
AND M_Os_Beweeg_Eiland_Omlaag  ; Merker One Shot Beweeg Eiland Omhoog
ANDNOT M_Arm_Omlaag  ; Merker Arm Omlaag Plc 1 & Plc 2
ANDNOT M_Delay_Arm_Omhoog  ; Merker Delay Arm Omhoog Plc 1 & Plc 2
ANDNOT MD_ARM_HAND  ; M_DYN_ARM DRUKKNOP
LD M_AUTO_BEDRIJF  ; Merker Auto Bedrijf
ANDNOT M_Show_Arm_Omhoog  ; Show Arm Omhoog
AND M_Show_Arm_Omlaag  ; Show Arm Omlaag
ORLD
AND M_Vrijgave_Arm_Beweging  ; Vrijgave Arm Mag Bewegen Plc 1 & Plc 2
SET Com1_Arm_Omlaag  ; PLC 1ARM OMLAAG
ANDNOT M_AUTO_BEDRIJF  ; Merker Auto Bedrijf
SET MD_ARM_HAND  ; M_DYN_ARM DRUKKNOP
; rung 5: Vertragen eiland op positie. / IOM Urs Schleapfer HvE 22-07-2010
LD P_On
AND I_42S10  ; EILAND OP POSITIE BENEDEN
TIM 0198 #20  ; Delay Eiland op positie (1.04)

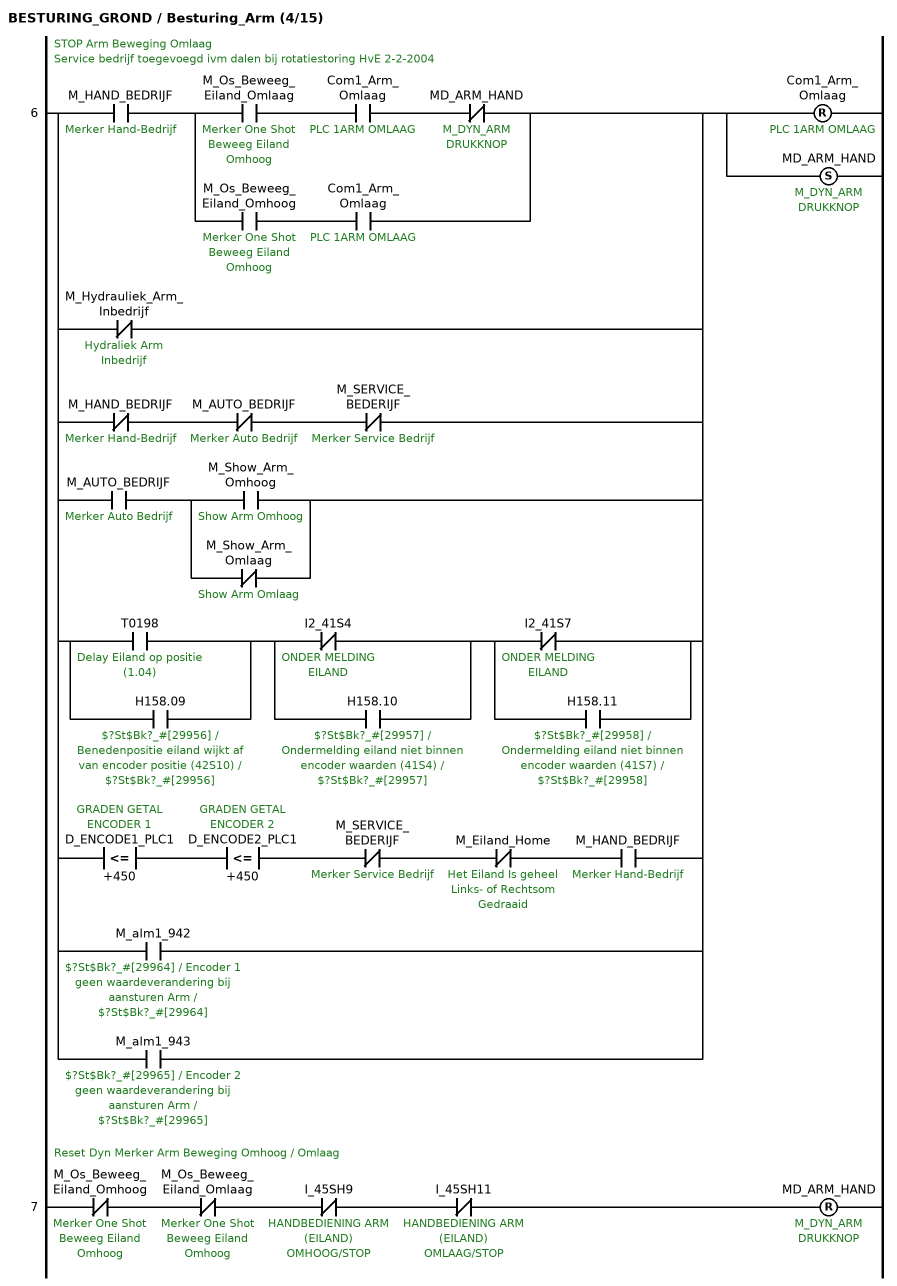
; rung 6: STOP Arm Beweging Omlaag / Service bedrijf toegevoegd ivm dalen bij rotatiestoring HvE 2-2-2004
LD M_HAND_BEDRIJF  ; Merker Hand-Bedrijf
LD M_Os_Beweeg_Eiland_Omlaag  ; Merker One Shot Beweeg Eiland Omhoog
AND Com1_Arm_Omlaag  ; PLC 1ARM OMLAAG
ANDNOT MD_ARM_HAND  ; M_DYN_ARM DRUKKNOP
LD M_Os_Beweeg_Eiland_Omhoog  ; Merker One Shot Beweeg Eiland Omhoog
AND Com1_Arm_Omlaag  ; PLC 1ARM OMLAAG
ORLD
ANDLD
ORNOT M_Hydrauliek_Arm_Inbedrijf  ; Hydraliek Arm Inbedrijf
LDNOT M_HAND_BEDRIJF  ; Merker Hand-Bedrijf
ANDNOT M_AUTO_BEDRIJF  ; Merker Auto Bedrijf
ANDNOT M_SERVICE_BEDERIJF  ; Merker Service Bedrijf
ORLD
LD M_AUTO_BEDRIJF  ; Merker Auto Bedrijf
LD M_Show_Arm_Omhoog  ; Show Arm Omhoog
ORNOT M_Show_Arm_Omlaag  ; Show Arm Omlaag
ANDLD
ORLD
LD T0198  ; Delay Eiland op positie (1.04)
OR H158.09  ; $?St$Bk?_#[29956] / Benedenpositie eiland wijkt af van encoder positie (42S10) / $?St$Bk?_#[29956]
LDNOT I2_41S4  ; ONDER MELDING EILAND
OR H158.10  ; $?St$Bk?_#[29957] / Ondermelding eiland niet binnen encoder waarden (41S4) / $?St$Bk?_#[29957]
ANDLD
LDNOT I2_41S7  ; ONDER MELDING EILAND
OR H158.11  ; $?St$Bk?_#[29958] / Ondermelding eiland niet binnen encoder waarden (41S7) / $?St$Bk?_#[29958]
ANDLD
ORLD
LD<=S(317) D_ENCODE1_PLC1 +450  ; GRADEN GETAL ENCODER 1
AND<=S(317) D_ENCODE2_PLC1 +450  ; GRADEN GETAL ENCODER 2
ANDNOT M_SERVICE_BEDERIJF  ; Merker Service Bedrijf
ANDNOT M_Eiland_Home  ; Het Eiland Is geheel Links- of Rechtsom Gedraaid
AND M_HAND_BEDRIJF  ; Merker Hand-Bedrijf
ORLD
OR M_alm1_942  ; $?St$Bk?_#[29964] / Encoder 1 geen waardeverandering bij aansturen Arm / $?St$Bk?_#[29964]
OR M_alm1_943  ; $?St$Bk?_#[29965] / Encoder 2 geen waardeverandering bij aansturen Arm / $?St$Bk?_#[29965]
RSET Com1_Arm_Omlaag  ; PLC 1ARM OMLAAG
SET MD_ARM_HAND  ; M_DYN_ARM DRUKKNOP
; rung 7: Reset Dyn Merker Arm Beweging Omhoog / Omlaag
LDNOT M_Os_Beweeg_Eiland_Omhoog  ; Merker One Shot Beweeg Eiland Omhoog
ANDNOT M_Os_Beweeg_Eiland_Omlaag  ; Merker One Shot Beweeg Eiland Omhoog
ANDNOT I_45SH9  ; HANDBEDIENING ARM (EILAND) OMHOOG/STOP
ANDNOT I_45SH11  ; HANDBEDIENING ARM (EILAND) OMLAAG/STOP
RSET MD_ARM_HAND  ; M_DYN_ARM DRUKKNOP

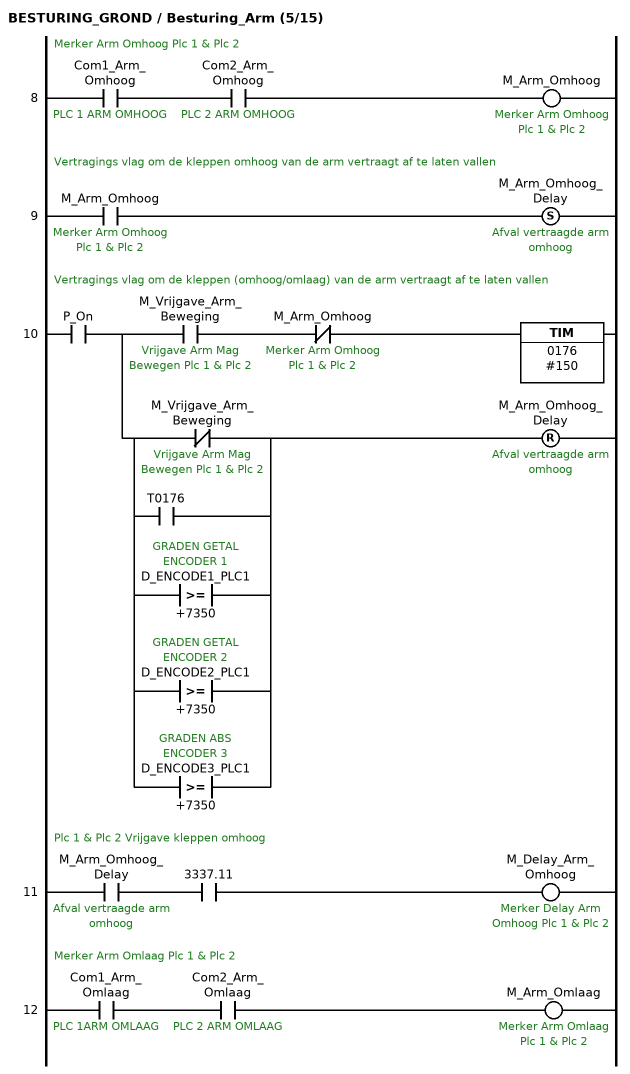
; rung 8: Merker Arm Omhoog Plc 1 & Plc 2
LD Com1_Arm_Omhoog  ; PLC 1 ARM OMHOOG
AND Com2_Arm_Omhoog  ; PLC 2 ARM OMHOOG
OUT M_Arm_Omhoog  ; Merker Arm Omhoog Plc 1 & Plc 2
; rung 9: Vertragings vlag om de kleppen omhoog van de arm vertraagt af te laten vallen
LD M_Arm_Omhoog  ; Merker Arm Omhoog Plc 1 & Plc 2
SET M_Arm_Omhoog_Delay  ; Afval vertraagde arm omhoog
; rung 10: Vertragings vlag om de kleppen (omhoog/omlaag) van de arm vertraagt af te laten vallen
LD P_On
OUT TR0
AND M_Vrijgave_Arm_Beweging  ; Vrijgave Arm Mag Bewegen Plc 1 & Plc 2
ANDNOT M_Arm_Omhoog  ; Merker Arm Omhoog Plc 1 & Plc 2
TIM 0176 #150
LD TR0
LDNOT M_Vrijgave_Arm_Beweging  ; Vrijgave Arm Mag Bewegen Plc 1 & Plc 2
OR T0176
OR>=S(327) D_ENCODE1_PLC1 +7350  ; GRADEN GETAL ENCODER 1
OR>=S(327) D_ENCODE2_PLC1 +7350  ; GRADEN GETAL ENCODER 2
OR>=S(327) D_ENCODE3_PLC1 +7350  ; GRADEN ABS ENCODER 3
ANDLD
RSET M_Arm_Omhoog_Delay  ; Afval vertraagde arm omhoog
; rung 11: Plc 1 & Plc 2 Vrijgave kleppen omhoog
LD M_Arm_Omhoog_Delay  ; Afval vertraagde arm omhoog
AND 3337.11
OUT M_Delay_Arm_Omhoog  ; Merker Delay Arm Omhoog Plc 1 & Plc 2
; rung 12: Merker Arm Omlaag Plc 1 & Plc 2
LD Com1_Arm_Omlaag  ; PLC 1ARM OMLAAG
AND Com2_Arm_Omlaag  ; PLC 2 ARM OMLAAG
OUT M_Arm_Omlaag  ; Merker Arm Omlaag Plc 1 & Plc 2

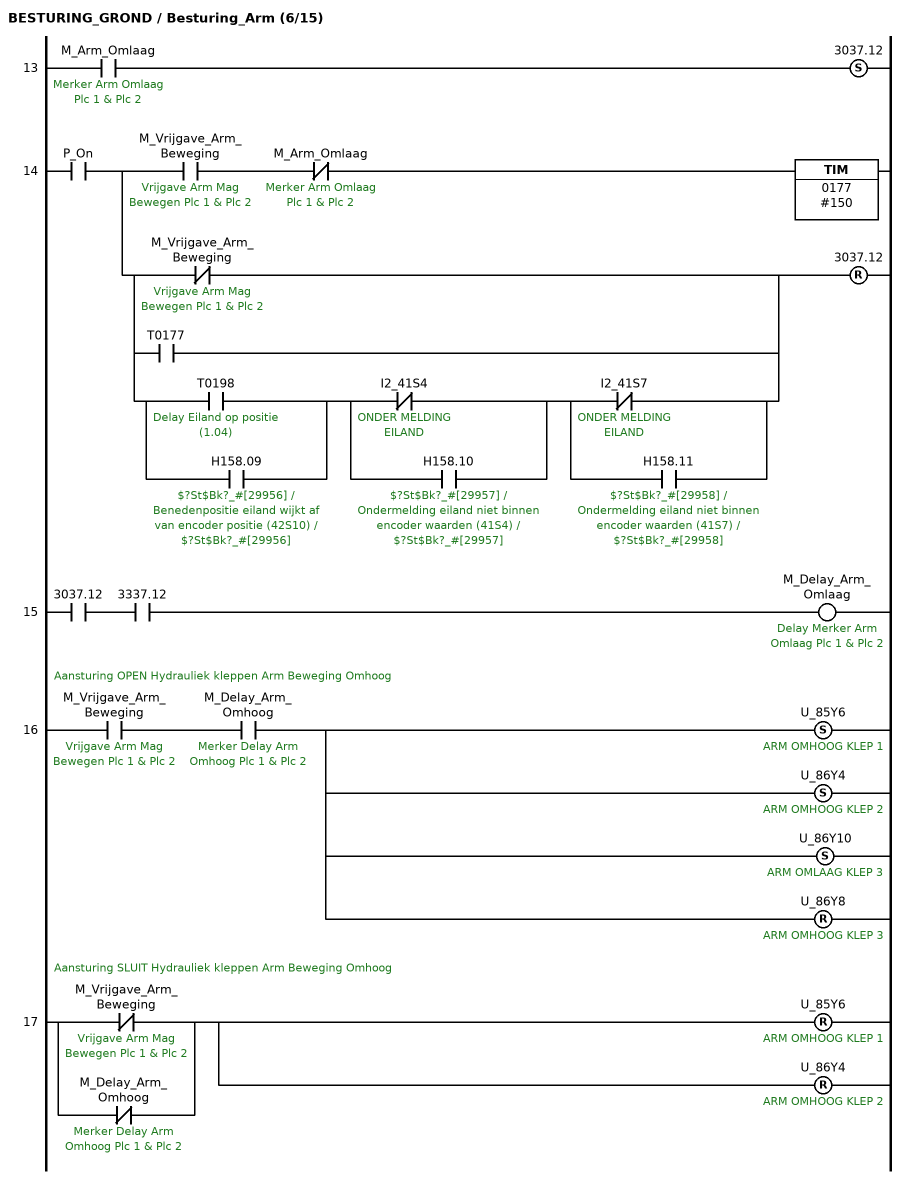
; rung 13
LD M_Arm_Omlaag  ; Merker Arm Omlaag Plc 1 & Plc 2
SET 3037.12
; rung 14
LD P_On
OUT TR0
AND M_Vrijgave_Arm_Beweging  ; Vrijgave Arm Mag Bewegen Plc 1 & Plc 2
ANDNOT M_Arm_Omlaag  ; Merker Arm Omlaag Plc 1 & Plc 2
TIM 0177 #150
LD TR0
LDNOT M_Vrijgave_Arm_Beweging  ; Vrijgave Arm Mag Bewegen Plc 1 & Plc 2
OR T0177
LD T0198  ; Delay Eiland op positie (1.04)
OR H158.09  ; $?St$Bk?_#[29956] / Benedenpositie eiland wijkt af van encoder positie (42S10) / $?St$Bk?_#[29956]
LDNOT I2_41S4  ; ONDER MELDING EILAND
OR H158.10  ; $?St$Bk?_#[29957] / Ondermelding eiland niet binnen encoder waarden (41S4) / $?St$Bk?_#[29957]
ANDLD
LDNOT I2_41S7  ; ONDER MELDING EILAND
OR H158.11  ; $?St$Bk?_#[29958] / Ondermelding eiland niet binnen encoder waarden (41S7) / $?St$Bk?_#[29958]
ANDLD
ORLD
ANDLD
RSET 3037.12
; rung 15
LD 3037.12
AND 3337.12
OUT M_Delay_Arm_Omlaag  ; Delay Merker Arm Omlaag Plc 1 & Plc 2
; rung 16: Aansturing OPEN Hydrauliek kleppen Arm Beweging Omhoog
LD M_Vrijgave_Arm_Beweging  ; Vrijgave Arm Mag Bewegen Plc 1 & Plc 2
AND M_Delay_Arm_Omhoog  ; Merker Delay Arm Omhoog Plc 1 & Plc 2
SET U_85Y6  ; ARM OMHOOG KLEP 1
SET U_86Y4  ; ARM OMHOOG KLEP 2
SET U_86Y10  ; ARM OMLAAG KLEP 3
RSET U_86Y8  ; ARM OMHOOG KLEP 3
; rung 17: Aansturing SLUIT Hydrauliek kleppen Arm Beweging Omhoog
LDNOT M_Vrijgave_Arm_Beweging  ; Vrijgave Arm Mag Bewegen Plc 1 & Plc 2
ORNOT M_Delay_Arm_Omhoog  ; Merker Delay Arm Omhoog Plc 1 & Plc 2
RSET U_85Y6  ; ARM OMHOOG KLEP 1
RSET U_86Y4  ; ARM OMHOOG KLEP 2

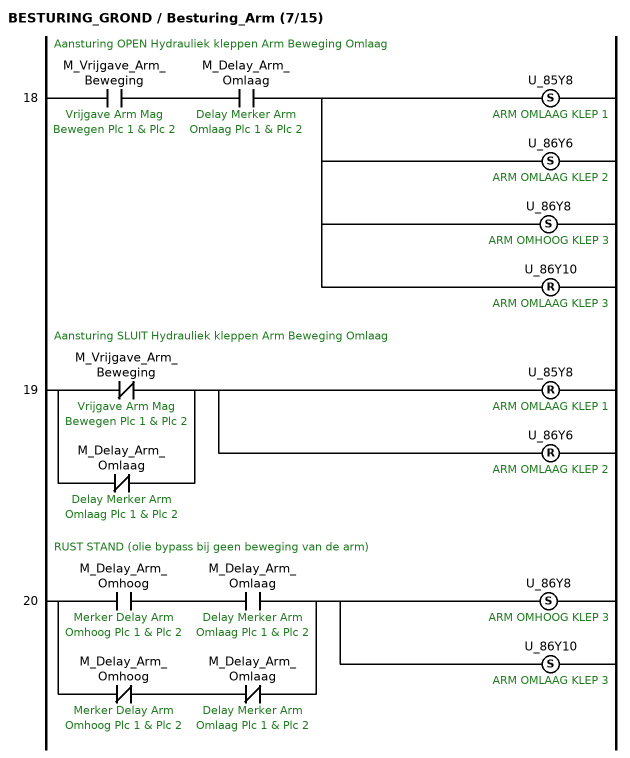
; rung 18: Aansturing OPEN Hydrauliek kleppen Arm Beweging Omlaag
LD M_Vrijgave_Arm_Beweging  ; Vrijgave Arm Mag Bewegen Plc 1 & Plc 2
AND M_Delay_Arm_Omlaag  ; Delay Merker Arm Omlaag Plc 1 & Plc 2
SET U_85Y8  ; ARM OMLAAG KLEP 1
SET U_86Y6  ; ARM OMLAAG KLEP 2
SET U_86Y8  ; ARM OMHOOG KLEP 3
RSET U_86Y10  ; ARM OMLAAG KLEP 3
; rung 19: Aansturing SLUIT Hydrauliek kleppen Arm Beweging Omlaag
LDNOT M_Vrijgave_Arm_Beweging  ; Vrijgave Arm Mag Bewegen Plc 1 & Plc 2
ORNOT M_Delay_Arm_Omlaag  ; Delay Merker Arm Omlaag Plc 1 & Plc 2
RSET U_85Y8  ; ARM OMLAAG KLEP 1
RSET U_86Y6  ; ARM OMLAAG KLEP 2
; rung 20: RUST STAND (olie bypass bij geen beweging van de arm)
LD M_Delay_Arm_Omhoog  ; Merker Delay Arm Omhoog Plc 1 & Plc 2
AND M_Delay_Arm_Omlaag  ; Delay Merker Arm Omlaag Plc 1 & Plc 2
LDNOT M_Delay_Arm_Omhoog  ; Merker Delay Arm Omhoog Plc 1 & Plc 2
ANDNOT M_Delay_Arm_Omlaag  ; Delay Merker Arm Omlaag Plc 1 & Plc 2
ORLD
SET U_86Y8  ; ARM OMHOOG KLEP 3
SET U_86Y10  ; ARM OMLAAG KLEP 3

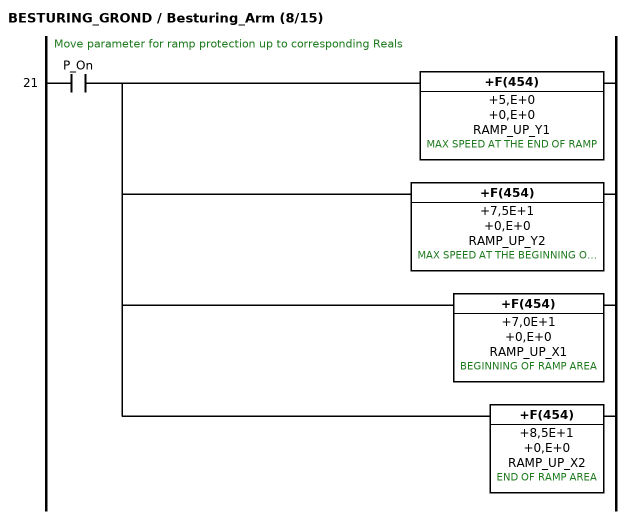
; rung 21: Move parameter for ramp protection up to corresponding Reals
LD P_On
+F(454) +5,E+0 +0,E+0 RAMP_UP_Y1  ; MAX SPEED AT THE END OF RAMP
+F(454) +7,5E+1 +0,E+0 RAMP_UP_Y2  ; MAX SPEED AT THE BEGINNING OF RAMP
+F(454) +7,0E+1 +0,E+0 RAMP_UP_X1  ; BEGINNING OF RAMP AREA
+F(454) +8,5E+1 +0,E+0 RAMP_UP_X2  ; END OF RAMP AREA

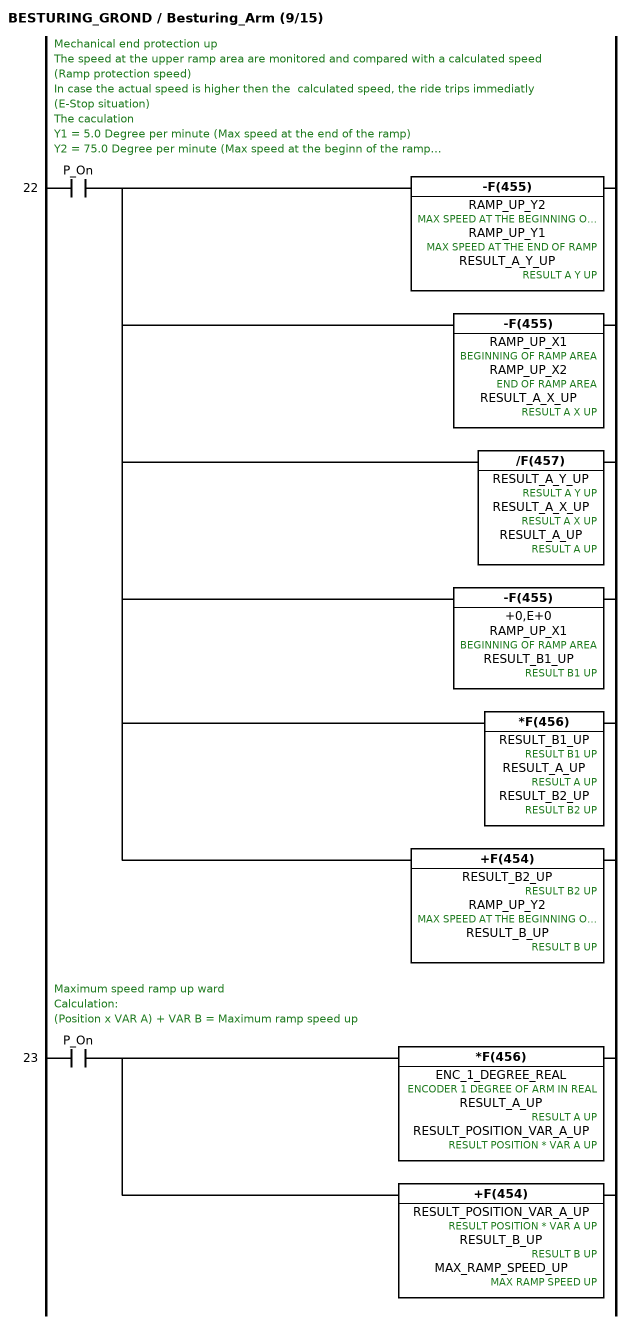
; rung 22: Mechanical end protection up / The speed at the upper ramp area are monitored and compared with a calculated speed (Ramp protection speed) / In case the actual speed is higher then the  calculated speed, the ride trips immediatly (E-Stop situation) / The caculation / Y1 = 5.0 Degree per minute (Max speed at the end of the ramp) / Y2 = 75.0 Degree per minute (Max speed at the beginn of the ramp) / X1 = 68.0 Degree (Begin of ramp area) / X2 = 85.0 Degree (End of ramp area) / The formula for A: / Y2 - Y1 / A =    ------- / X1 - X2 / The formula for B: / B =    (A * (0 - X1) + Y2
LD P_On
-F(455) RAMP_UP_Y2 RAMP_UP_Y1 RESULT_A_Y_UP  ; MAX SPEED AT THE BEGINNING OF RAMP, MAX SPEED AT THE END OF RAMP, RESULT A Y UP
-F(455) RAMP_UP_X1 RAMP_UP_X2 RESULT_A_X_UP  ; BEGINNING OF RAMP AREA, END OF RAMP AREA, RESULT A X UP
/F(457) RESULT_A_Y_UP RESULT_A_X_UP RESULT_A_UP  ; RESULT A Y UP, RESULT A X UP, RESULT A UP
-F(455) +0,E+0 RAMP_UP_X1 RESULT_B1_UP  ; BEGINNING OF RAMP AREA, RESULT B1 UP
*F(456) RESULT_B1_UP RESULT_A_UP RESULT_B2_UP  ; RESULT B1 UP, RESULT A UP, RESULT B2 UP
+F(454) RESULT_B2_UP RAMP_UP_Y2 RESULT_B_UP  ; RESULT B2 UP, MAX SPEED AT THE BEGINNING OF RAMP, RESULT B UP
; rung 23: Maximum speed ramp up ward / Calculation: / (Position x VAR A) + VAR B = Maximum ramp speed up
LD P_On
*F(456) ENC_1_DEGREE_REAL RESULT_A_UP RESULT_POSITION_VAR_A_UP  ; ENCODER 1 DEGREE OF ARM IN REAL, RESULT A UP, RESULT POSITION * VAR A UP
+F(454) RESULT_POSITION_VAR_A_UP RESULT_B_UP MAX_RAMP_SPEED_UP  ; RESULT POSITION * VAR A UP, RESULT B UP, MAX RAMP SPEED UP

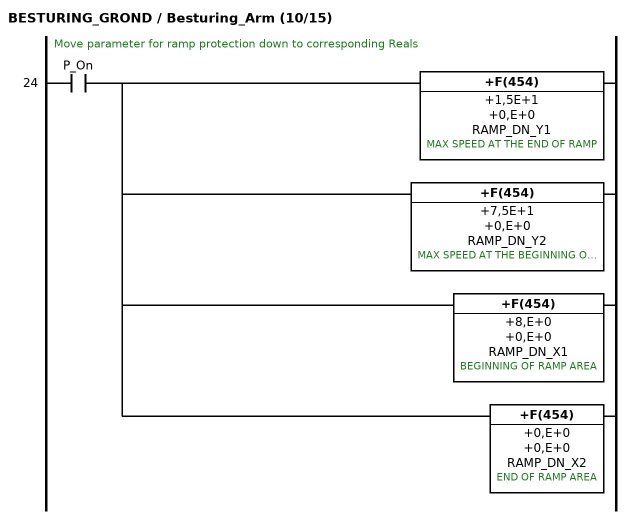
; rung 24: Move parameter for ramp protection down to corresponding Reals
LD P_On
+F(454) +1,5E+1 +0,E+0 RAMP_DN_Y1  ; MAX SPEED AT THE END OF RAMP
+F(454) +7,5E+1 +0,E+0 RAMP_DN_Y2  ; MAX SPEED AT THE BEGINNING OF RAMP
+F(454) +8,E+0 +0,E+0 RAMP_DN_X1  ; BEGINNING OF RAMP AREA
+F(454) +0,E+0 +0,E+0 RAMP_DN_X2  ; END OF RAMP AREA

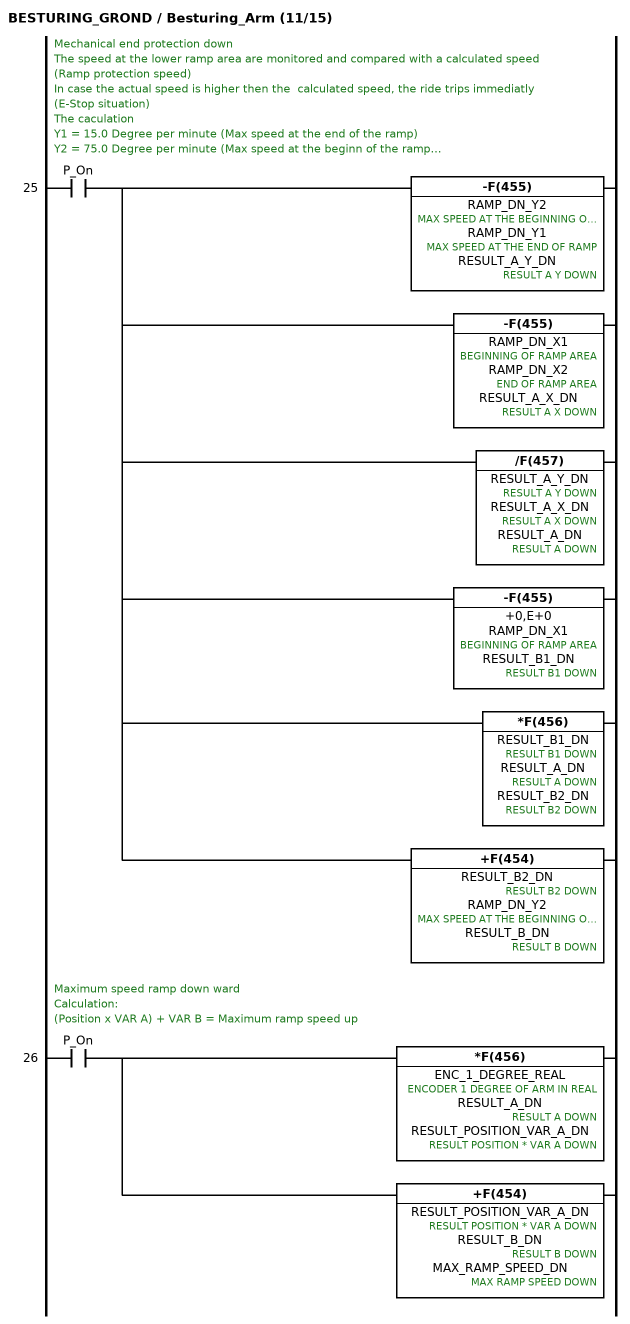
; rung 25: Mechanical end protection down / The speed at the lower ramp area are monitored and compared with a calculated speed (Ramp protection speed) / In case the actual speed is higher then the  calculated speed, the ride trips immediatly (E-Stop situation) / The caculation / Y1 = 15.0 Degree per minute (Max speed at the end of the ramp) / Y2 = 75.0 Degree per minute (Max speed at the beginn of the ramp) / X1 = 8.0 Degree (Begin of ramp area) / X2 = 0.0 Degree (End of ramp area) / The formula for A: / Y2 - Y1 / A =    ------- / X1 - X2 / The formula for B: / B =    (A * (0 - X1) + Y2
LD P_On
-F(455) RAMP_DN_Y2 RAMP_DN_Y1 RESULT_A_Y_DN  ; MAX SPEED AT THE BEGINNING OF RAMP, MAX SPEED AT THE END OF RAMP, RESULT A Y DOWN
-F(455) RAMP_DN_X1 RAMP_DN_X2 RESULT_A_X_DN  ; BEGINNING OF RAMP AREA, END OF RAMP AREA, RESULT A X DOWN
/F(457) RESULT_A_Y_DN RESULT_A_X_DN RESULT_A_DN  ; RESULT A Y DOWN, RESULT A X DOWN, RESULT A DOWN
-F(455) +0,E+0 RAMP_DN_X1 RESULT_B1_DN  ; BEGINNING OF RAMP AREA, RESULT B1 DOWN
*F(456) RESULT_B1_DN RESULT_A_DN RESULT_B2_DN  ; RESULT B1 DOWN, RESULT A DOWN, RESULT B2 DOWN
+F(454) RESULT_B2_DN RAMP_DN_Y2 RESULT_B_DN  ; RESULT B2 DOWN, MAX SPEED AT THE BEGINNING OF RAMP, RESULT B DOWN
; rung 26: Maximum speed ramp down ward / Calculation: / (Position x VAR A) + VAR B = Maximum ramp speed up
LD P_On
*F(456) ENC_1_DEGREE_REAL RESULT_A_DN RESULT_POSITION_VAR_A_DN  ; ENCODER 1 DEGREE OF ARM IN REAL, RESULT A DOWN, RESULT POSITION * VAR A DOWN
+F(454) RESULT_POSITION_VAR_A_DN RESULT_B_DN MAX_RAMP_SPEED_DN  ; RESULT POSITION * VAR A DOWN, RESULT B DOWN, MAX RAMP SPEED DOWN

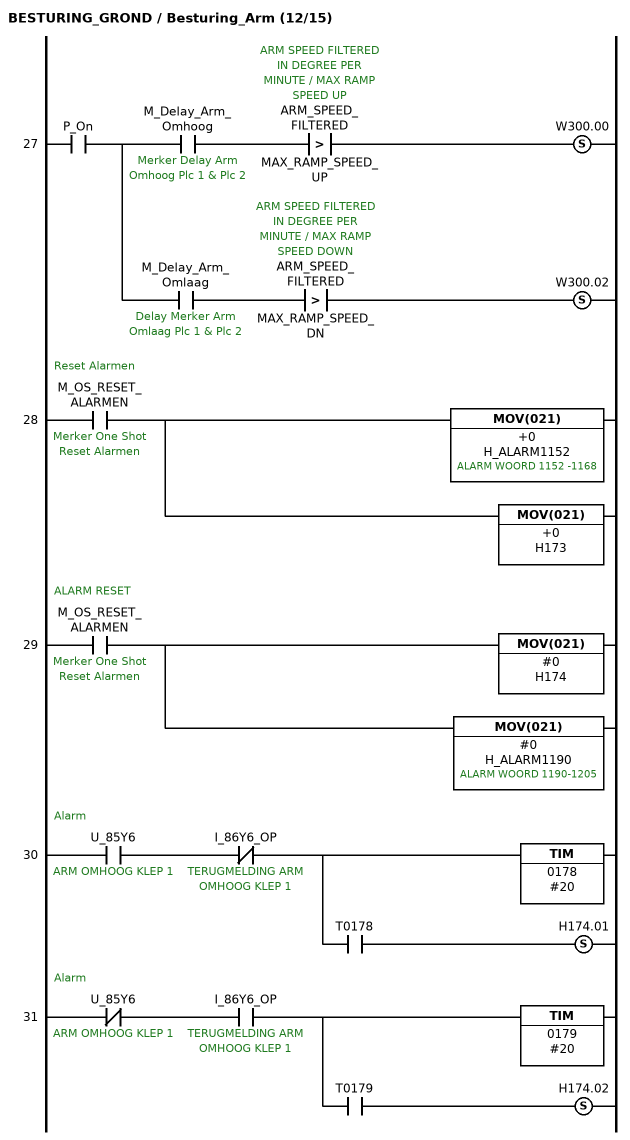
; rung 27
LD P_On
OUT TR0
AND M_Delay_Arm_Omhoog  ; Merker Delay Arm Omhoog Plc 1 & Plc 2
AND>F(333) ARM_SPEED_FILTERED MAX_RAMP_SPEED_UP  ; ARM SPEED FILTERED IN DEGREE PER MINUTE, MAX RAMP SPEED UP
SET W300.00
LD TR0
AND M_Delay_Arm_Omlaag  ; Delay Merker Arm Omlaag Plc 1 & Plc 2
AND>F(333) ARM_SPEED_FILTERED MAX_RAMP_SPEED_DN  ; ARM SPEED FILTERED IN DEGREE PER MINUTE, MAX RAMP SPEED DOWN
SET W300.02
; rung 28: Reset Alarmen
LD M_OS_RESET_ALARMEN  ; Merker One Shot Reset Alarmen
MOV(021) +0 H_ALARM1152  ; ALARM WOORD 1152 -1168
MOV(021) +0 H173
; rung 29: ALARM RESET
LD M_OS_RESET_ALARMEN  ; Merker One Shot Reset Alarmen
MOV(021) #0 H174
MOV(021) #0 H_ALARM1190  ; ALARM WOORD 1190-1205
; rung 30: Alarm
LD U_85Y6  ; ARM OMHOOG KLEP 1
ANDNOT I_86Y6_OP  ; TERUGMELDING ARM OMHOOG KLEP 1
TIM 0178 #20
AND T0178
SET H174.01
; rung 31: Alarm
LDNOT U_85Y6  ; ARM OMHOOG KLEP 1
AND I_86Y6_OP  ; TERUGMELDING ARM OMHOOG KLEP 1
TIM 0179 #20
AND T0179
SET H174.02

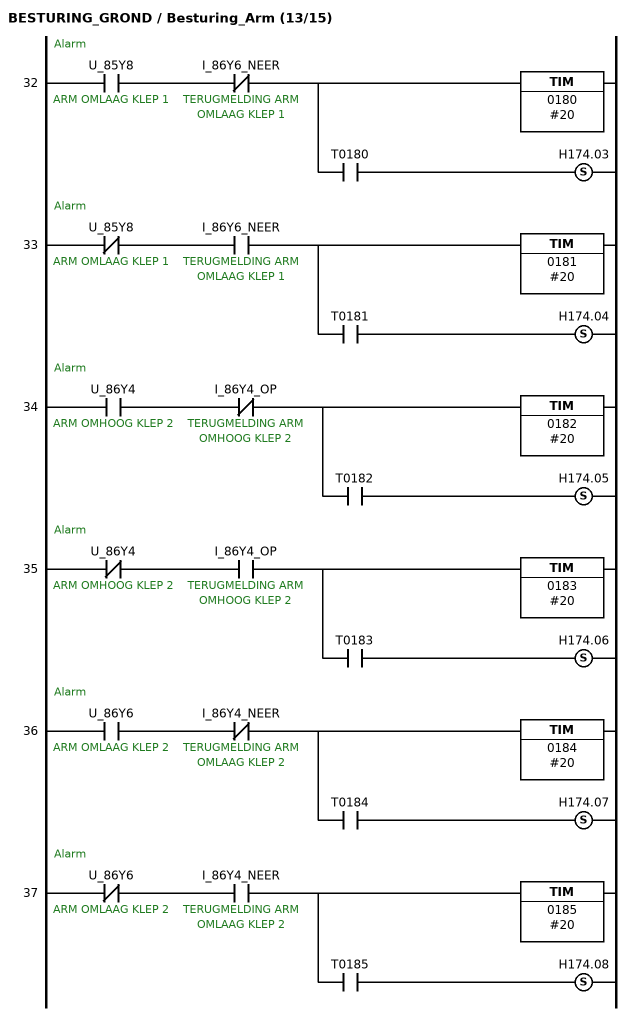
; rung 32: Alarm
LD U_85Y8  ; ARM OMLAAG KLEP 1
ANDNOT I_86Y6_NEER  ; TERUGMELDING ARM OMLAAG KLEP 1
TIM 0180 #20
AND T0180
SET H174.03
; rung 33: Alarm
LDNOT U_85Y8  ; ARM OMLAAG KLEP 1
AND I_86Y6_NEER  ; TERUGMELDING ARM OMLAAG KLEP 1
TIM 0181 #20
AND T0181
SET H174.04
; rung 34: Alarm
LD U_86Y4  ; ARM OMHOOG KLEP 2
ANDNOT I_86Y4_OP  ; TERUGMELDING ARM OMHOOG KLEP 2
TIM 0182 #20
AND T0182
SET H174.05
; rung 35: Alarm
LDNOT U_86Y4  ; ARM OMHOOG KLEP 2
AND I_86Y4_OP  ; TERUGMELDING ARM OMHOOG KLEP 2
TIM 0183 #20
AND T0183
SET H174.06
; rung 36: Alarm
LD U_86Y6  ; ARM OMLAAG KLEP 2
ANDNOT I_86Y4_NEER  ; TERUGMELDING ARM OMLAAG KLEP 2
TIM 0184 #20
AND T0184
SET H174.07
; rung 37: Alarm
LDNOT U_86Y6  ; ARM OMLAAG KLEP 2
AND I_86Y4_NEER  ; TERUGMELDING ARM OMLAAG KLEP 2
TIM 0185 #20
AND T0185
SET H174.08

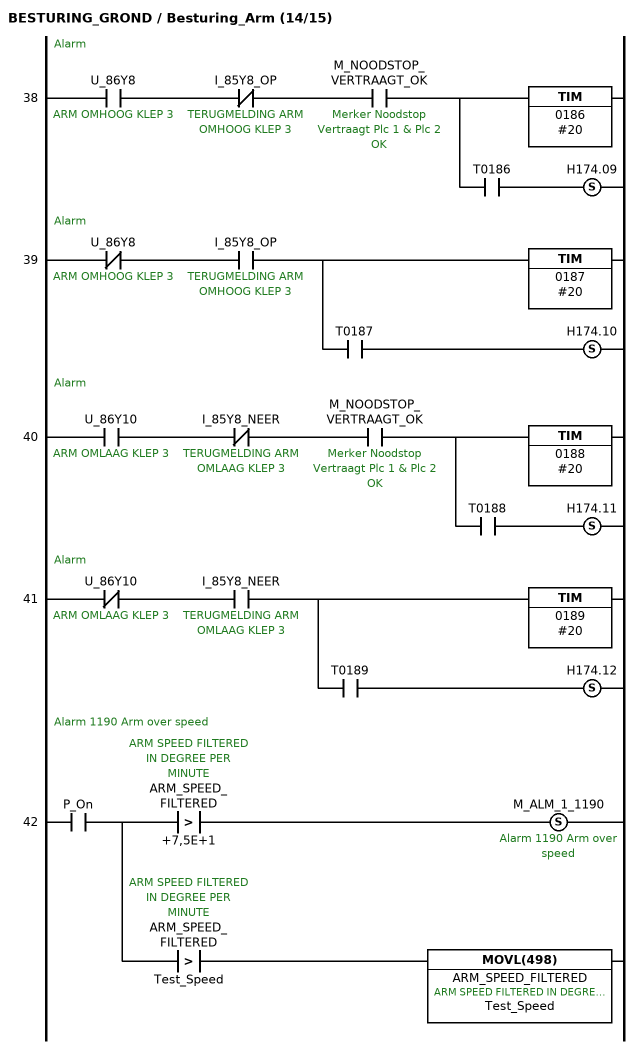
; rung 38: Alarm
LD U_86Y8  ; ARM OMHOOG KLEP 3
ANDNOT I_85Y8_OP  ; TERUGMELDING ARM OMHOOG KLEP 3
AND M_NOODSTOP_VERTRAAGT_OK  ; Merker Noodstop Vertraagt Plc 1 & Plc 2 OK
TIM 0186 #20
AND T0186
SET H174.09
; rung 39: Alarm
LDNOT U_86Y8  ; ARM OMHOOG KLEP 3
AND I_85Y8_OP  ; TERUGMELDING ARM OMHOOG KLEP 3
TIM 0187 #20
AND T0187
SET H174.10
; rung 40: Alarm
LD U_86Y10  ; ARM OMLAAG KLEP 3
ANDNOT I_85Y8_NEER  ; TERUGMELDING ARM OMLAAG KLEP 3
AND M_NOODSTOP_VERTRAAGT_OK  ; Merker Noodstop Vertraagt Plc 1 & Plc 2 OK
TIM 0188 #20
AND T0188
SET H174.11
; rung 41: Alarm
LDNOT U_86Y10  ; ARM OMLAAG KLEP 3
AND I_85Y8_NEER  ; TERUGMELDING ARM OMLAAG KLEP 3
TIM 0189 #20
AND T0189
SET H174.12
; rung 42: Alarm 1190 Arm over speed
LD P_On
OUT TR0
AND>F(333) ARM_SPEED_FILTERED +7,5E+1  ; ARM SPEED FILTERED IN DEGREE PER MINUTE
SET M_ALM_1_1190  ; Alarm 1190 Arm over speed
LD TR0
AND>F(333) ARM_SPEED_FILTERED Test_Speed  ; ARM SPEED FILTERED IN DEGREE PER MINUTE
MOVL(498) ARM_SPEED_FILTERED Test_Speed  ; ARM SPEED FILTERED IN DEGREE PER MINUTE

